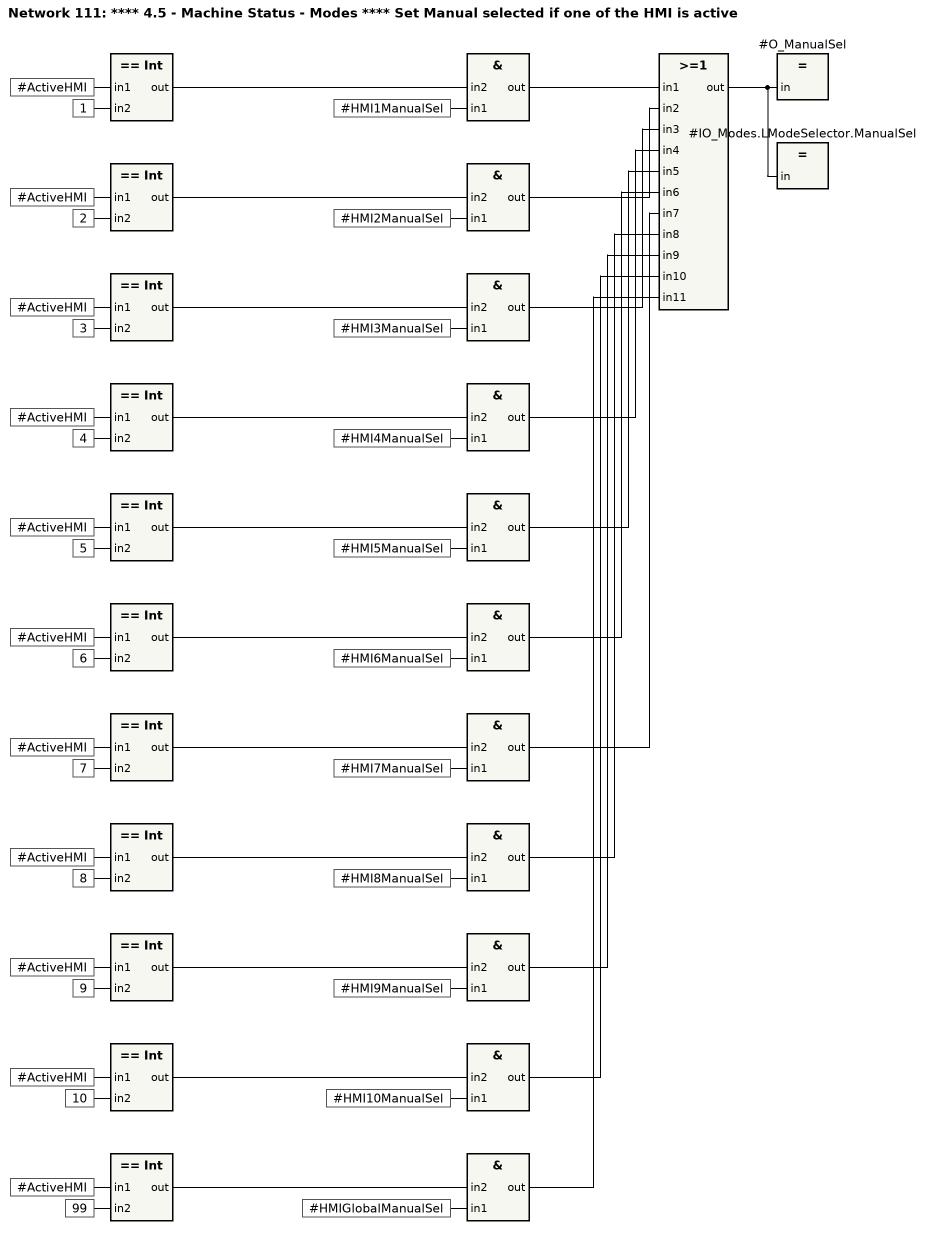
   #O_ManualSel := ((#ActiveHMI = 1) AND #HMI1ManualSel) OR ((#ActiveHMI = 2) AND #HMI2ManualSel) OR ((#ActiveHMI = 3) AND #HMI3ManualSel) OR ((#ActiveHMI = 4) AND #HMI4ManualSel) OR ((#ActiveHMI = 5) AND #HMI5ManualSel) OR ((#ActiveHMI = 6) AND #HMI6ManualSel) OR ((#ActiveHMI = 7) AND #HMI7ManualSel) OR ((#ActiveHMI = 8) AND #HMI8ManualSel) OR ((#ActiveHMI = 9) AND #HMI9ManualSel) OR ((#ActiveHMI = 10) AND #HMI10ManualSel) OR ((#ActiveHMI = 99) AND #HMIGlobalManualSel);
   #IO_Modes.LModeSelector.ManualSel := #O_ManualSel;
END_REGION

REGION Network 112: **** 4.6 - Machine Status - Indications **** Animation
   // Animation
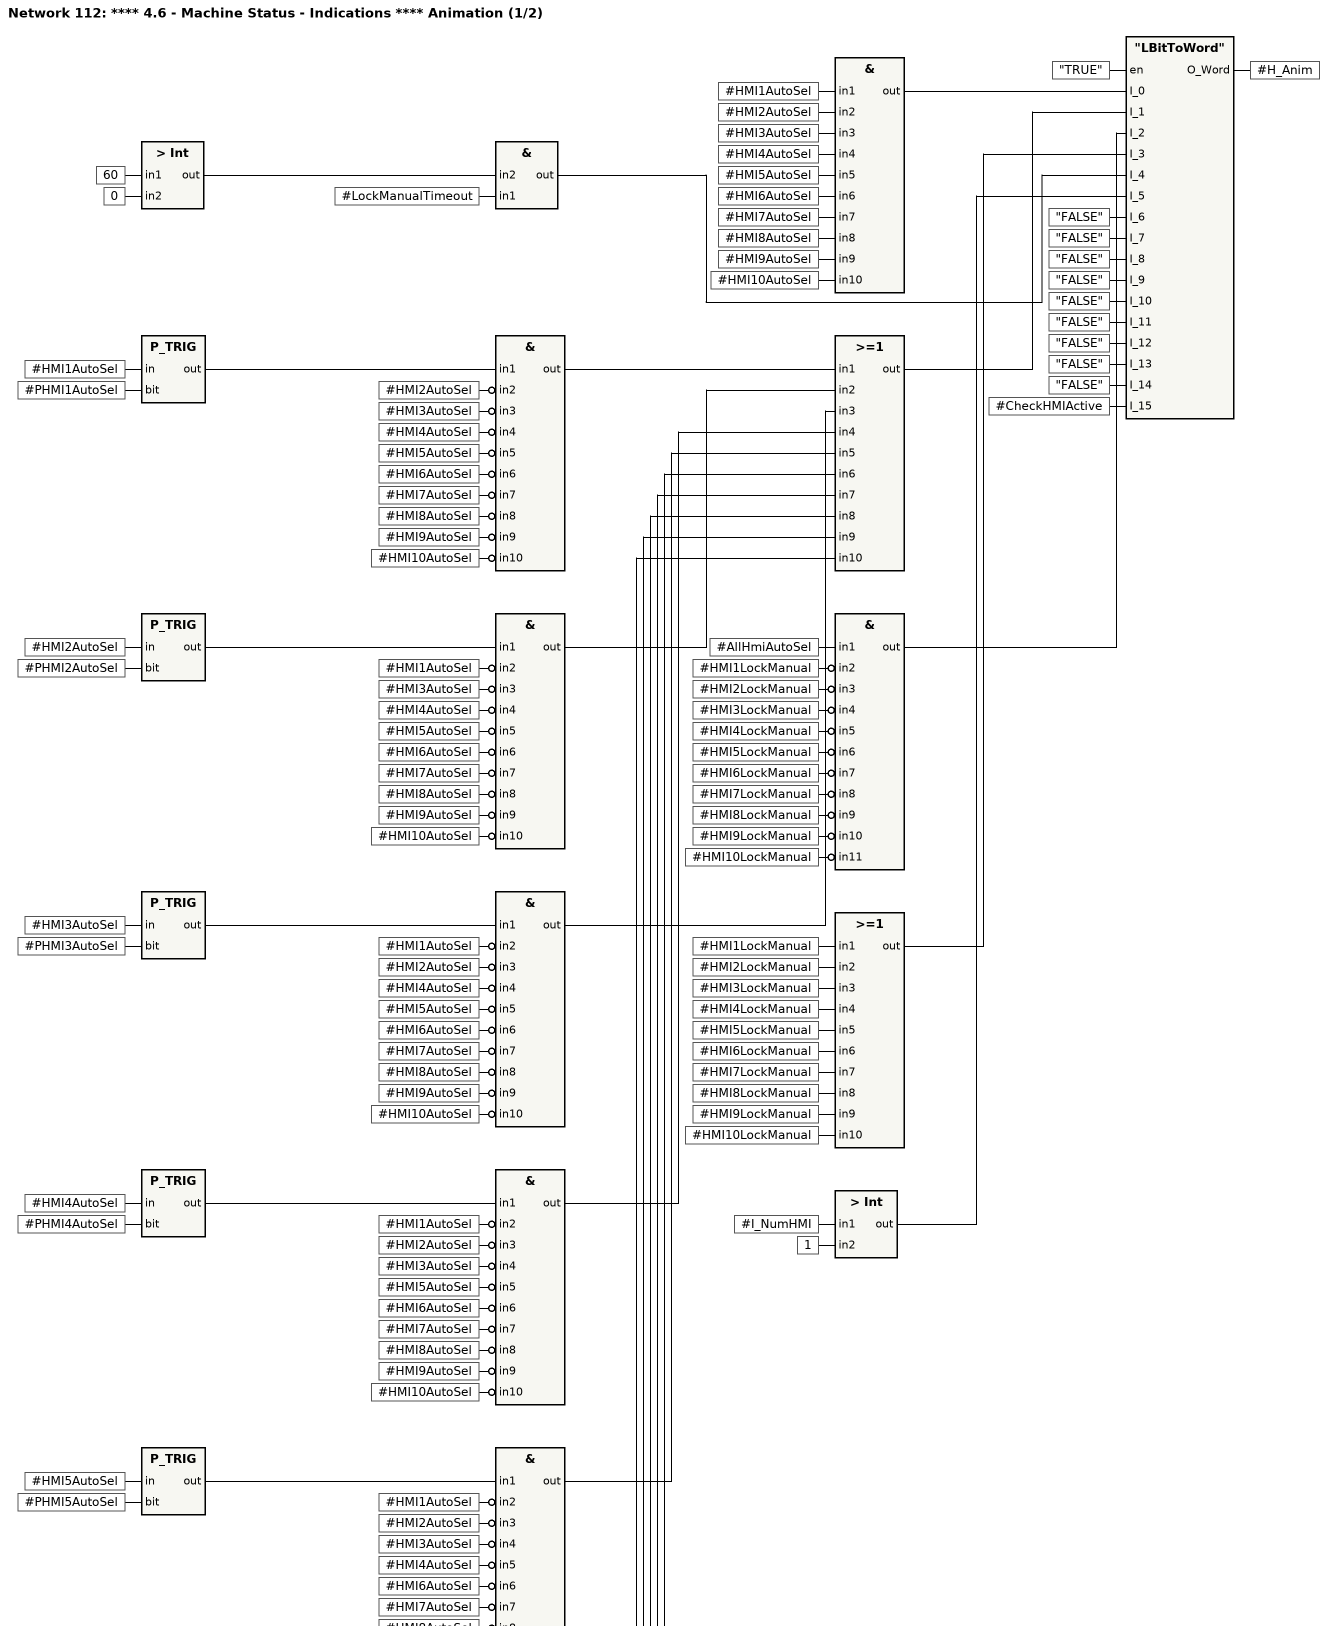
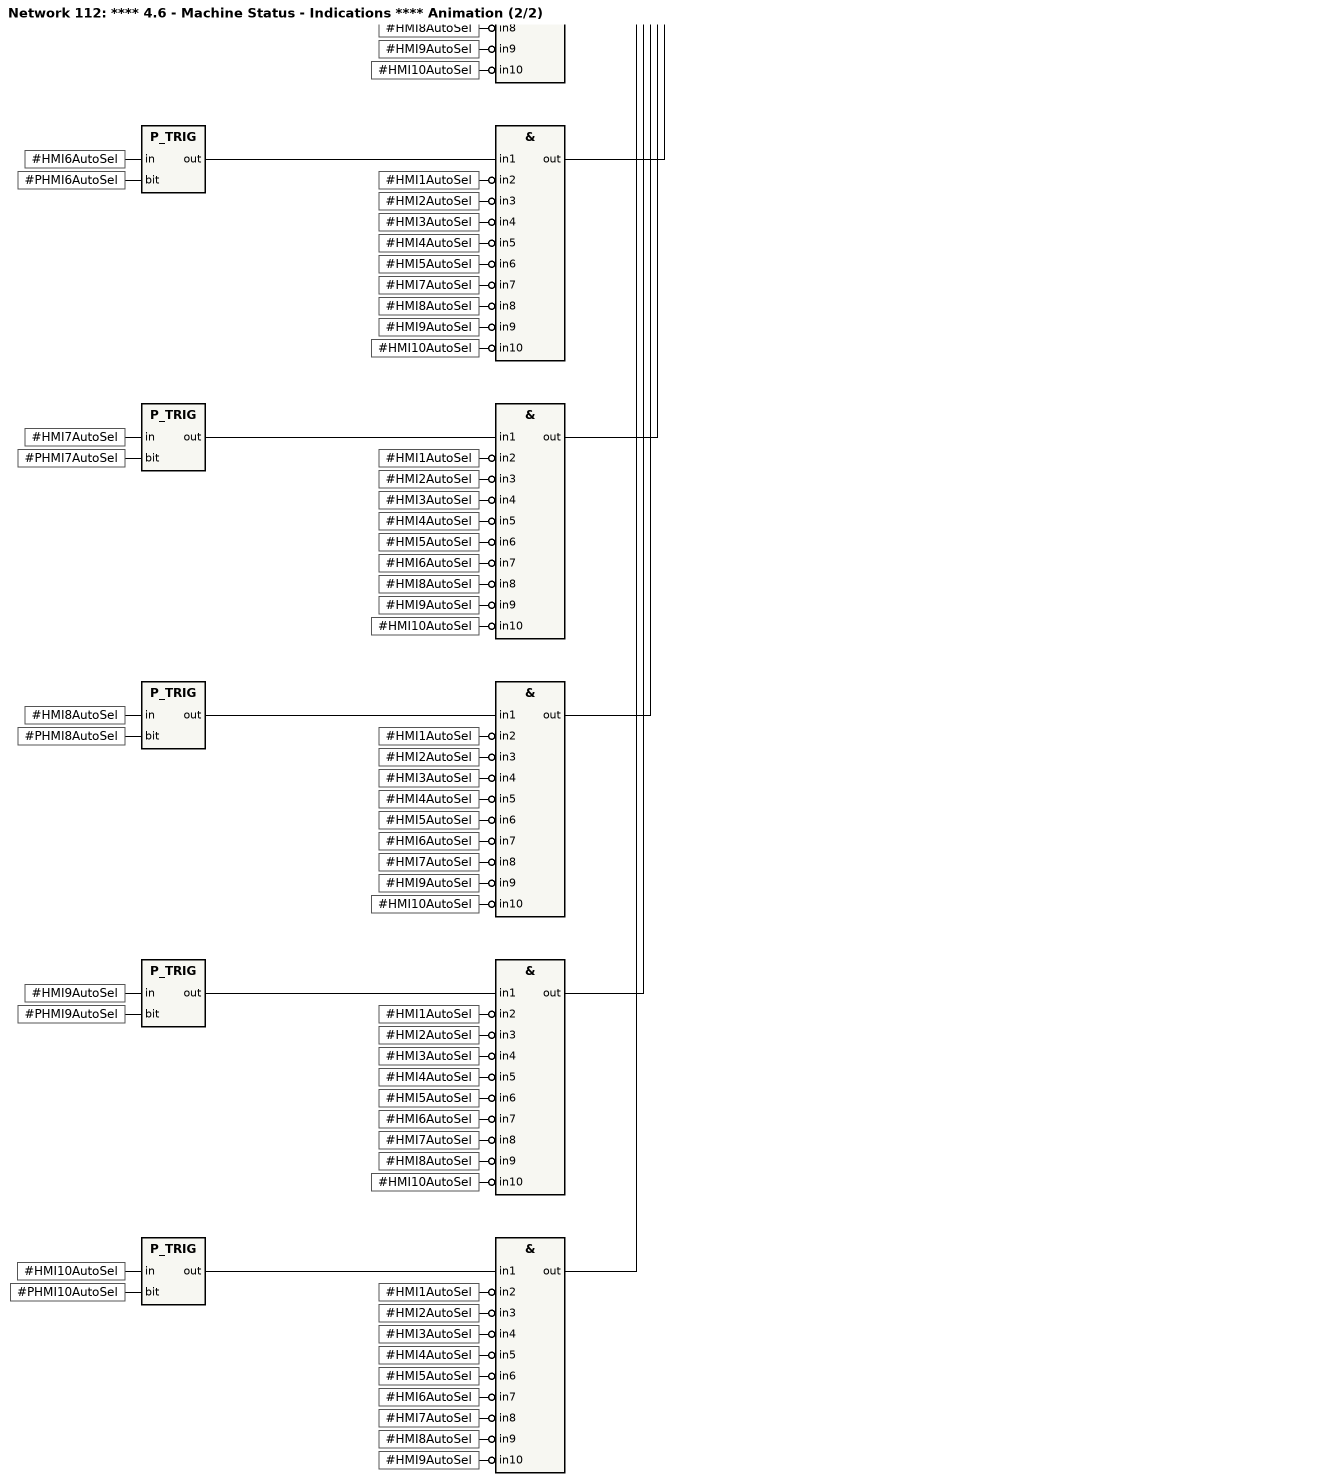
   #_w1 := #HMI1AutoSel AND NOT #PHMI1AutoSel;   // rising edge
   #PHMI1AutoSel := #HMI1AutoSel;
   #_w2 := #HMI2AutoSel AND NOT #PHMI2AutoSel;   // rising edge
   #PHMI2AutoSel := #HMI2AutoSel;
   #_w3 := #HMI3AutoSel AND NOT #PHMI3AutoSel;   // rising edge
   #PHMI3AutoSel := #HMI3AutoSel;
   #_w4 := #HMI4AutoSel AND NOT #PHMI4AutoSel;   // rising edge
   #PHMI4AutoSel := #HMI4AutoSel;
   #_w5 := #HMI5AutoSel AND NOT #PHMI5AutoSel;   // rising edge
   #PHMI5AutoSel := #HMI5AutoSel;
   #_w6 := #HMI6AutoSel AND NOT #PHMI6AutoSel;   // rising edge
   #PHMI6AutoSel := #HMI6AutoSel;
   #_w7 := #HMI7AutoSel AND NOT #PHMI7AutoSel;   // rising edge
   #PHMI7AutoSel := #HMI7AutoSel;
   #_w8 := #HMI8AutoSel AND NOT #PHMI8AutoSel;   // rising edge
   #PHMI8AutoSel := #HMI8AutoSel;
   #_w9 := #HMI9AutoSel AND NOT #PHMI9AutoSel;   // rising edge
   #PHMI9AutoSel := #HMI9AutoSel;
   #_w10 := #HMI10AutoSel AND NOT #PHMI10AutoSel;   // rising edge
   #PHMI10AutoSel := #HMI10AutoSel;
   IF "TRUE" THEN
       "LBitToWord"(I_0 := #HMI1AutoSel AND #HMI2AutoSel AND #HMI3AutoSel AND #HMI4AutoSel AND #HMI5AutoSel AND #HMI6AutoSel AND #HMI7AutoSel AND #HMI8AutoSel AND #HMI9AutoSel AND #HMI10AutoSel,
                    I_1 := (#_w1 AND NOT #HMI2AutoSel AND NOT #HMI3AutoSel AND NOT #HMI4AutoSel AND NOT #HMI5AutoSel AND NOT #HMI6AutoSel AND NOT #HMI7AutoSel AND NOT #HMI8AutoSel AND NOT #HMI9AutoSel AND NOT #HMI10AutoSel) OR (#_w2 AND NOT #HMI1AutoSel AND NOT #HMI3AutoSel AND NOT #HMI4AutoSel AND NOT #HMI5AutoSel AND NOT #HMI6AutoSel AND NOT #HMI7AutoSel AND NOT #HMI8AutoSel AND NOT #HMI9AutoSel AND NOT #HMI10AutoSel) OR (#_w3 AND NOT #HMI1AutoSel AND NOT #HMI2AutoSel AND NOT #HMI4AutoSel AND NOT #HMI5AutoSel AND NOT #HMI6AutoSel AND NOT #HMI7AutoSel AND NOT #HMI8AutoSel AND NOT #HMI9AutoSel AND NOT #HMI10AutoSel) OR (#_w4 AND NOT #HMI1AutoSel AND NOT #HMI2AutoSel AND NOT #HMI3AutoSel AND NOT #HMI5AutoSel AND NOT #HMI6AutoSel AND NOT #HMI7AutoSel AND NOT #HMI8AutoSel AND NOT #HMI9AutoSel AND NOT #HMI10AutoSel) OR (#_w5 AND NOT #HMI1AutoSel AND NOT #HMI2AutoSel AND NOT #HMI3AutoSel AND NOT #HMI4AutoSel AND NOT #HMI6AutoSel AND NOT #HMI7AutoSel AND NOT #HMI8AutoSel AND NOT #HMI9AutoSel AND NOT #HMI10AutoSel) OR (#_w6 AND NOT #HMI1AutoSel AND NOT #HMI2AutoSel AND NOT #HMI3AutoSel AND NOT #HMI4AutoSel AND NOT #HMI5AutoSel AND NOT #HMI7AutoSel AND NOT #HMI8AutoSel AND NOT #HMI9AutoSel AND NOT #HMI10AutoSel) OR (#_w7 AND NOT #HMI1AutoSel AND NOT #HMI2AutoSel AND NOT #HMI3AutoSel AND NOT #HMI4AutoSel AND NOT #HMI5AutoSel AND NOT #HMI6AutoSel AND NOT #HMI8AutoSel AND NOT #HMI9AutoSel AND NOT #HMI10AutoSel) OR (#_w8 AND NOT #HMI1AutoSel AND NOT #HMI2AutoSel AND NOT #HMI3AutoSel AND NOT #HMI4AutoSel AND NOT #HMI5AutoSel AND NOT #HMI6AutoSel AND NOT #HMI7AutoSel AND NOT #HMI9AutoSel AND NOT #HMI10AutoSel) OR (#_w9 AND NOT #HMI1AutoSel AND NOT #HMI2AutoSel AND NOT #HMI3AutoSel AND NOT #HMI4AutoSel AND NOT #HMI5AutoSel AND NOT #HMI6AutoSel AND NOT #HMI7AutoSel AND NOT #HMI8AutoSel AND NOT #HMI10AutoSel) OR (#_w10 AND NOT #HMI1AutoSel AND NOT #HMI2AutoSel AND NOT #HMI3AutoSel AND NOT #HMI4AutoSel AND NOT #HMI5AutoSel AND NOT #HMI6AutoSel AND NOT #HMI7AutoSel AND NOT #HMI8AutoSel AND NOT #HMI9AutoSel),
                    I_2 := #AllHmiAutoSel AND NOT #HMI1LockManual AND NOT #HMI2LockManual AND NOT #HMI3LockManual AND NOT #HMI4LockManual AND NOT #HMI5LockManual AND NOT #HMI6LockManual AND NOT #HMI7LockManual AND NOT #HMI8LockManual AND NOT #HMI9LockManual AND NOT #HMI10LockManual,
                    I_3 := #HMI1LockManual OR #HMI2LockManual OR #HMI3LockManual OR #HMI4LockManual OR #HMI5LockManual OR #HMI6LockManual OR #HMI7LockManual OR #HMI8LockManual OR #HMI9LockManual OR #HMI10LockManual,
                    I_4 := (60 > 0) AND #LockManualTimeout,
                    I_5 := #I_NumHMI > 1,
                    I_6 := "FALSE",
                    I_7 := "FALSE",
                    I_8 := "FALSE",
                    I_9 := "FALSE",
                    I_10 := "FALSE",
                    I_11 := "FALSE",
                    I_12 := "FALSE",
                    I_13 := "FALSE",
                    I_14 := "FALSE",
                    I_15 := #CheckHMIActive,
                    O_Word => #H_Anim);
   END_IF;
END_REGION

REGION Network 113: **** 5.2 - Equations - Flow **** Reset transport memory on active HMI
   // Reset transport memory on active HMI
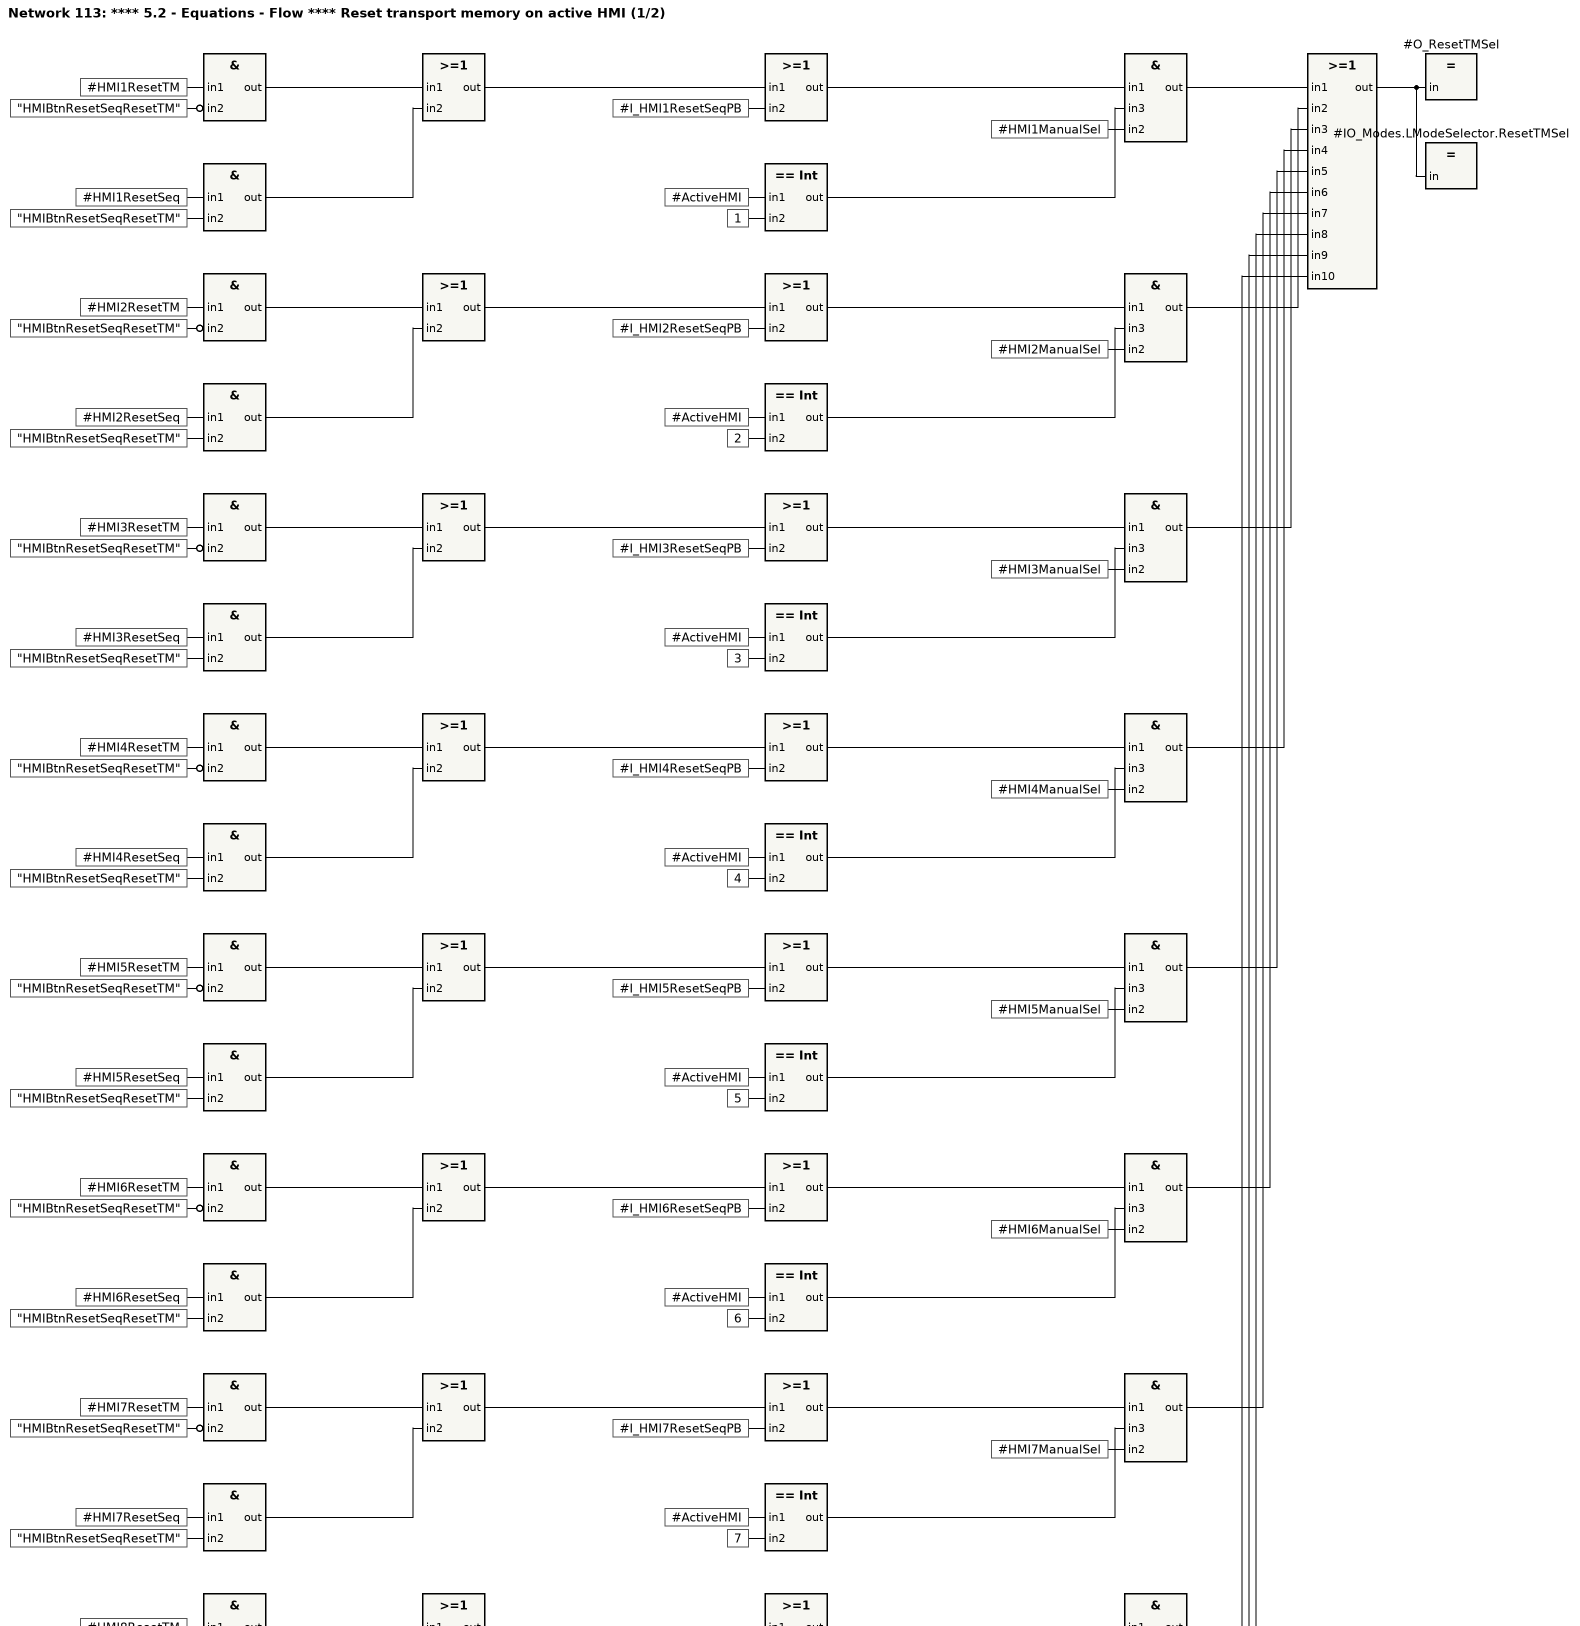
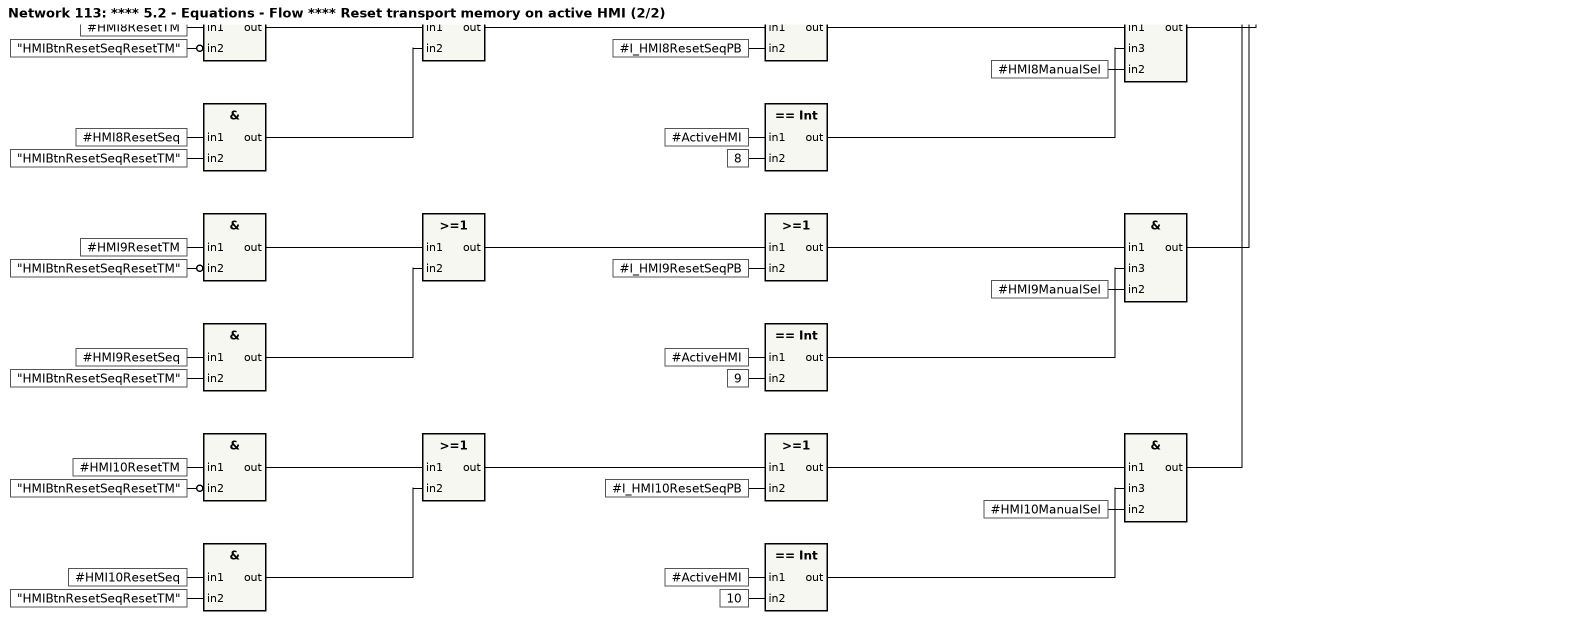
   #O_ResetTMSel := (((#HMI1ResetTM AND NOT "HMIBtnResetSeqResetTM") OR (#HMI1ResetSeq AND "HMIBtnResetSeqResetTM") OR #I_HMI1ResetSeqPB) AND (#ActiveHMI = 1) AND #HMI1ManualSel) OR (((#HMI2ResetTM AND NOT "HMIBtnResetSeqResetTM") OR (#HMI2ResetSeq AND "HMIBtnResetSeqResetTM") OR #I_HMI2ResetSeqPB) AND (#ActiveHMI = 2) AND #HMI2ManualSel) OR (((#HMI3ResetTM AND NOT "HMIBtnResetSeqResetTM") OR (#HMI3ResetSeq AND "HMIBtnResetSeqResetTM") OR #I_HMI3ResetSeqPB) AND (#ActiveHMI = 3) AND #HMI3ManualSel) OR (((#HMI4ResetTM AND NOT "HMIBtnResetSeqResetTM") OR (#HMI4ResetSeq AND "HMIBtnResetSeqResetTM") OR #I_HMI4ResetSeqPB) AND (#ActiveHMI = 4) AND #HMI4ManualSel) OR (((#HMI5ResetTM AND NOT "HMIBtnResetSeqResetTM") OR (#HMI5ResetSeq AND "HMIBtnResetSeqResetTM") OR #I_HMI5ResetSeqPB) AND (#ActiveHMI = 5) AND #HMI5ManualSel) OR (((#HMI6ResetTM AND NOT "HMIBtnResetSeqResetTM") OR (#HMI6ResetSeq AND "HMIBtnResetSeqResetTM") OR #I_HMI6ResetSeqPB) AND (#ActiveHMI = 6) AND #HMI6ManualSel) OR (((#HMI7ResetTM AND NOT "HMIBtnResetSeqResetTM") OR (#HMI7ResetSeq AND "HMIBtnResetSeqResetTM") OR #I_HMI7ResetSeqPB) AND (#ActiveHMI = 7) AND #HMI7ManualSel) OR (((#HMI8ResetTM AND NOT "HMIBtnResetSeqResetTM") OR (#HMI8ResetSeq AND "HMIBtnResetSeqResetTM") OR #I_HMI8ResetSeqPB) AND (#ActiveHMI = 8) AND #HMI8ManualSel) OR (((#HMI9ResetTM AND NOT "HMIBtnResetSeqResetTM") OR (#HMI9ResetSeq AND "HMIBtnResetSeqResetTM") OR #I_HMI9ResetSeqPB) AND (#ActiveHMI = 9) AND #HMI9ManualSel) OR (((#HMI10ResetTM AND NOT "HMIBtnResetSeqResetTM") OR (#HMI10ResetSeq AND "HMIBtnResetSeqResetTM") OR #I_HMI10ResetSeqPB) AND (#ActiveHMI = 10) AND #HMI10ManualSel);
   #IO_Modes.LModeSelector.ResetTMSel := #O_ResetTMSel;
END_REGION

REGION Network 114: **** 5.2 - Equations - Flow **** Reset sequence on active HMI
   // Reset sequence on active HMI
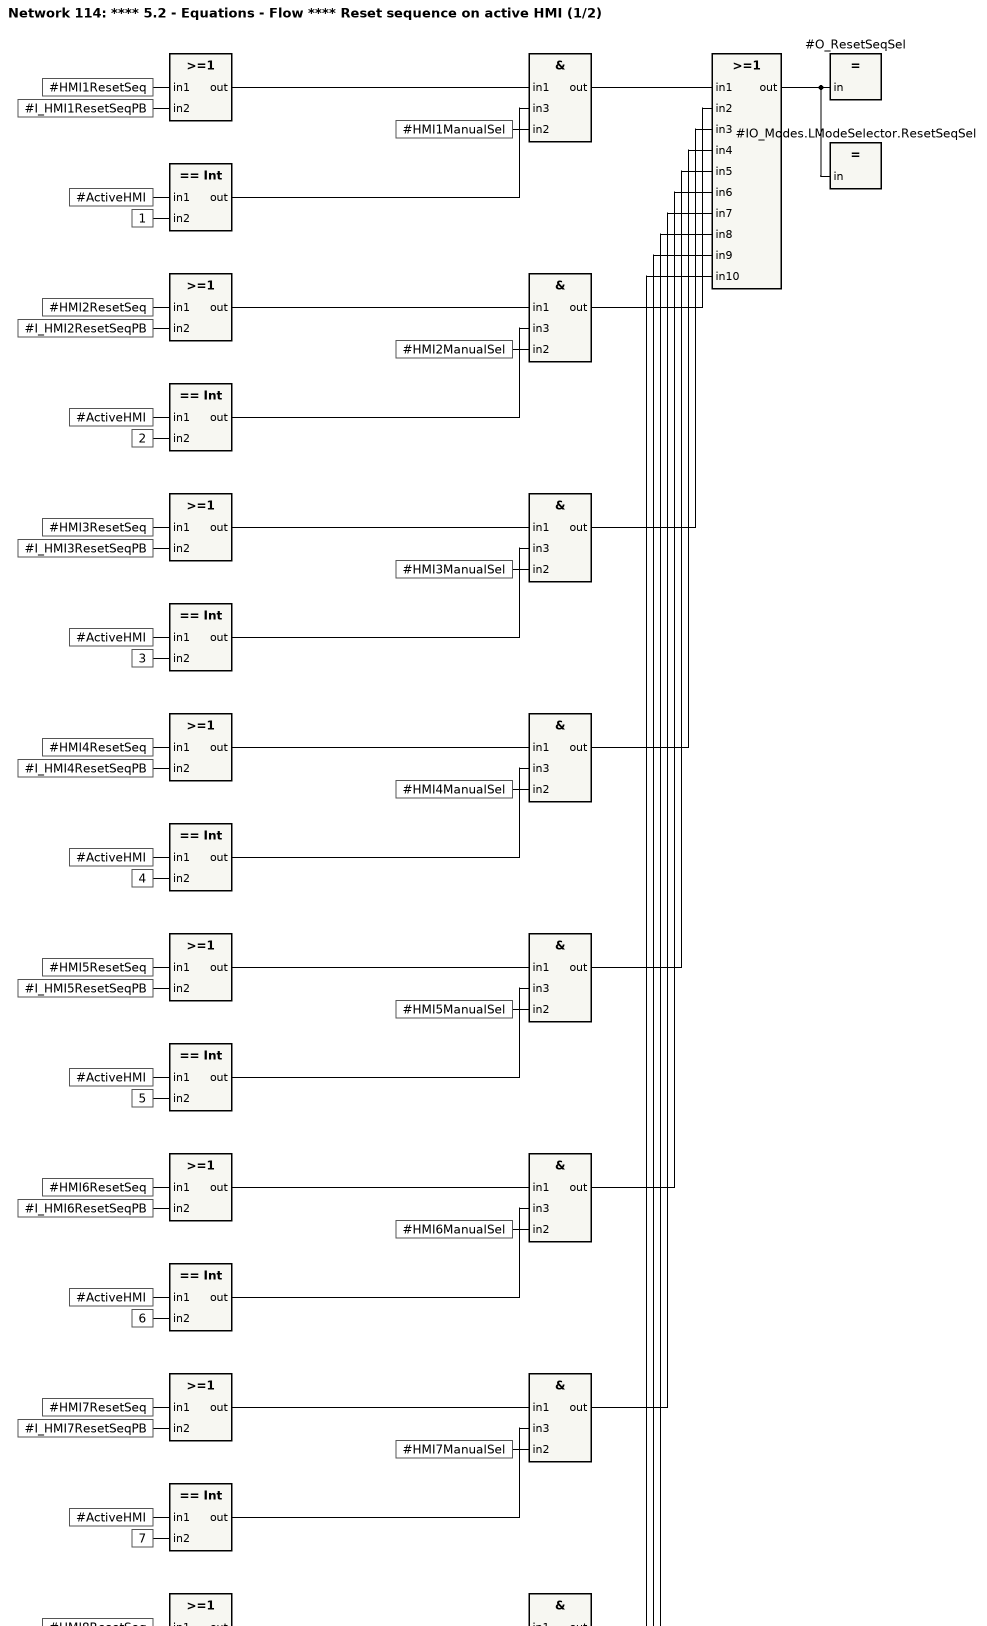
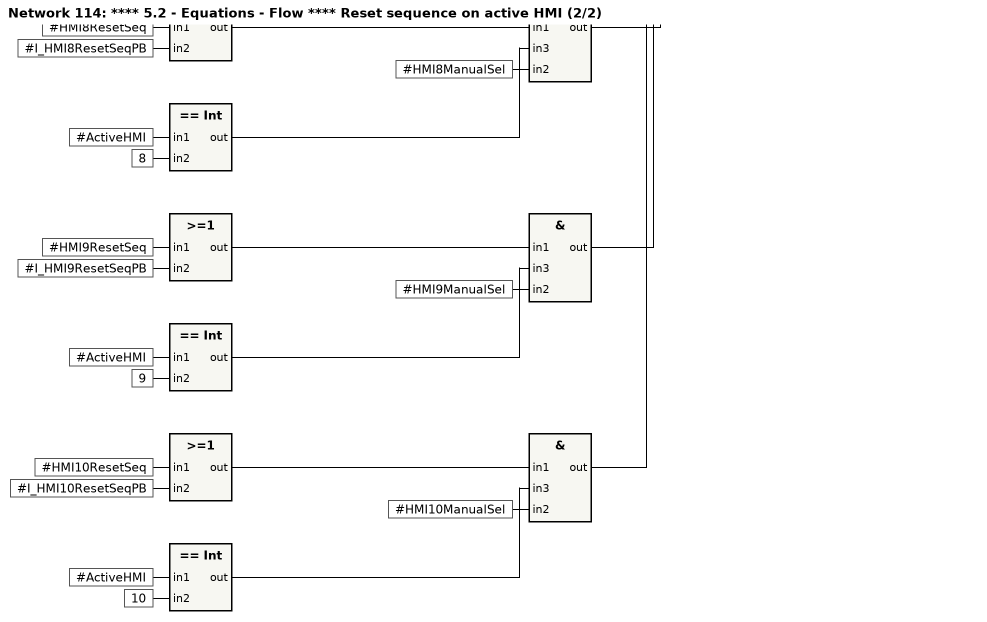
   #O_ResetSeqSel := ((#HMI1ResetSeq OR #I_HMI1ResetSeqPB) AND (#ActiveHMI = 1) AND #HMI1ManualSel) OR ((#HMI2ResetSeq OR #I_HMI2ResetSeqPB) AND (#ActiveHMI = 2) AND #HMI2ManualSel) OR ((#HMI3ResetSeq OR #I_HMI3ResetSeqPB) AND (#ActiveHMI = 3) AND #HMI3ManualSel) OR ((#HMI4ResetSeq OR #I_HMI4ResetSeqPB) AND (#ActiveHMI = 4) AND #HMI4ManualSel) OR ((#HMI5ResetSeq OR #I_HMI5ResetSeqPB) AND (#ActiveHMI = 5) AND #HMI5ManualSel) OR ((#HMI6ResetSeq OR #I_HMI6ResetSeqPB) AND (#ActiveHMI = 6) AND #HMI6ManualSel) OR ((#HMI7ResetSeq OR #I_HMI7ResetSeqPB) AND (#ActiveHMI = 7) AND #HMI7ManualSel) OR ((#HMI8ResetSeq OR #I_HMI8ResetSeqPB) AND (#ActiveHMI = 8) AND #HMI8ManualSel) OR ((#HMI9ResetSeq OR #I_HMI9ResetSeqPB) AND (#ActiveHMI = 9) AND #HMI9ManualSel) OR ((#HMI10ResetSeq OR #I_HMI10ResetSeqPB) AND (#ActiveHMI = 10) AND #HMI10ManualSel);
   #IO_Modes.LModeSelector.ResetSeqSel := #O_ResetSeqSel;
END_REGION

REGION Network 115: **** 5.2 - Equations - Flow **** Check Active HMI again - HMI <> 0
   // Check Active HMI again
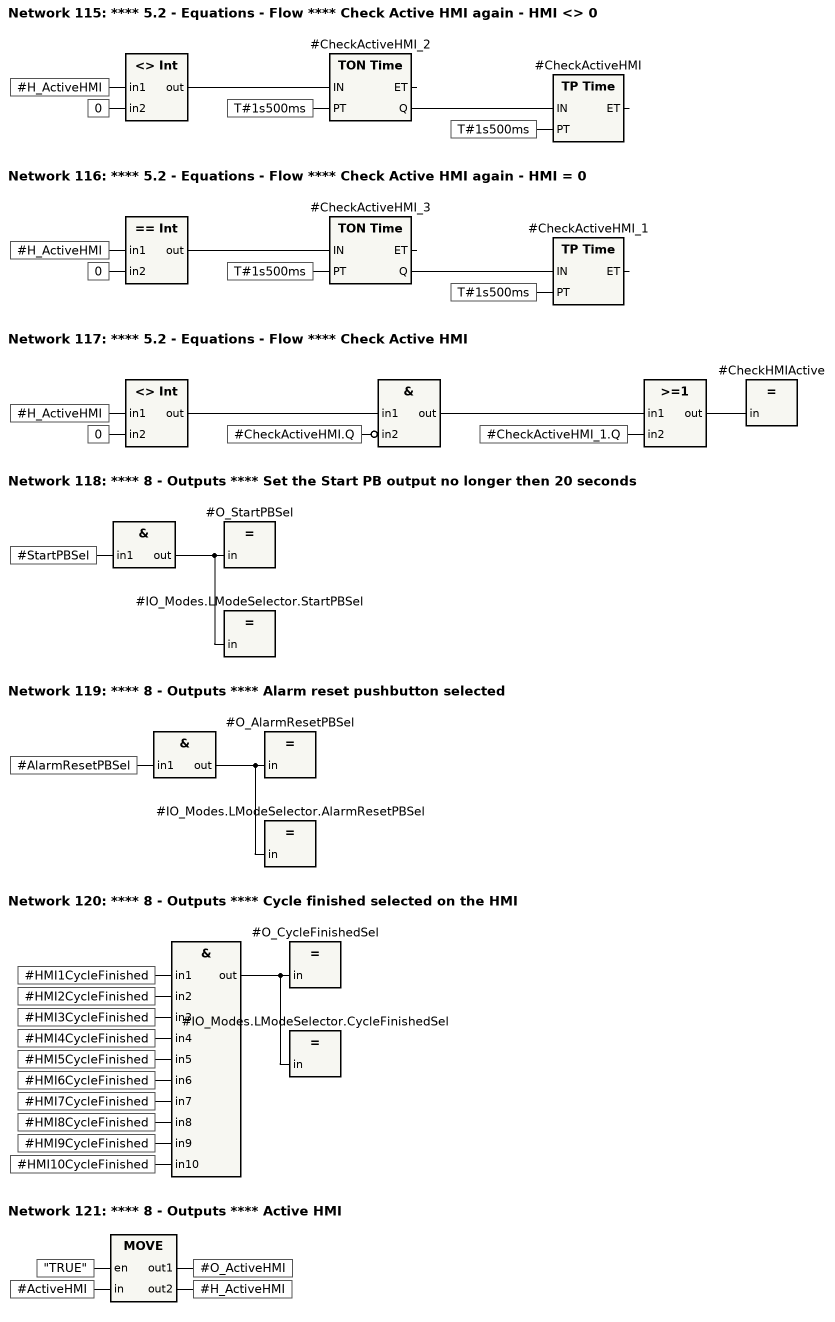
   #CheckActiveHMI_2(IN := #H_ActiveHMI <> 0, PT := T#1s500ms);   // TON
   #CheckActiveHMI(IN := #CheckActiveHMI_2.Q, PT := T#1s500ms);   // TP
END_REGION

REGION Network 116: **** 5.2 - Equations - Flow **** Check Active HMI again - HMI = 0
   // Check Active HMI again
   #CheckActiveHMI_3(IN := #H_ActiveHMI = 0, PT := T#1s500ms);   // TON
   #CheckActiveHMI_1(IN := #CheckActiveHMI_3.Q, PT := T#1s500ms);   // TP
END_REGION

REGION Network 117: **** 5.2 - Equations - Flow **** Check Active HMI
   // Check Active HMI
   #CheckHMIActive := ((#H_ActiveHMI <> 0) AND NOT #CheckActiveHMI.Q) OR #CheckActiveHMI_1.Q;
END_REGION

REGION Network 118: **** 8 - Outputs **** Set the Start PB output no longer then 20 seconds
   // Set the Start PB output no longer then 20 seconds
   #O_StartPBSel := #StartPBSel;
   #IO_Modes.LModeSelector.StartPBSel := #StartPBSel;
END_REGION

REGION Network 119: **** 8 - Outputs **** Alarm reset pushbutton selected
   // Alarm reset pushbutton selected
   #O_AlarmResetPBSel := #AlarmResetPBSel;
   #IO_Modes.LModeSelector.AlarmResetPBSel := #AlarmResetPBSel;
END_REGION

REGION Network 120: **** 8 - Outputs **** Cycle finished selected on the HMI
   // Cycle finished selected on the HMI
   #O_CycleFinishedSel := #HMI1CycleFinished AND #HMI2CycleFinished AND #HMI3CycleFinished AND #HMI4CycleFinished AND #HMI5CycleFinished AND #HMI6CycleFinished AND #HMI7CycleFinished AND #HMI8CycleFinished AND #HMI9CycleFinished AND #HMI10CycleFinished;
   #IO_Modes.LModeSelector.CycleFinishedSel := #O_CycleFinishedSel;
END_REGION

REGION Network 121: **** 8 - Outputs **** Active HMI
   // Active HMI
   IF "TRUE" THEN
       #O_ActiveHMI := #ActiveHMI;
       #H_ActiveHMI := #ActiveHMI;
   END_IF;
END_REGION

REGION Network 122: **** 8 - Outputs **** Lock Manual Time
   // Lock Manual Time
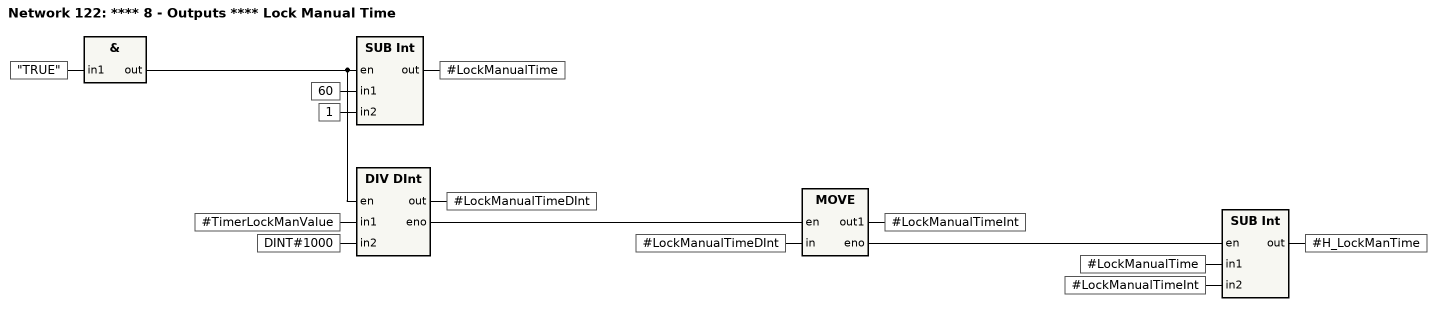
   // ENO of a box is taken as its EN; it also drops when the box reports an error
   IF "TRUE" THEN
       #LockManualTime := 60 - 1;
       #LockManualTimeDInt := #TimerLockManValue / DINT#1000;
       #LockManualTimeInt := #LockManualTimeDInt;
       #H_LockManTime := #LockManualTime - #LockManualTimeInt;
   END_IF;
END_REGION
END_FUNCTION_BLOCK

FUNCTION_BLOCK "LHMIResetStart"   // FB1006, FBD
TITLE = LHMIResetStart
{ S7_Optimized_Access := 'FALSE' }
AUTHOR : VCC
FAMILY : Control
NAME : ModeSel
VERSION : 1.0
// ================================================================================
// This module is creating the needed integers for the F_ACK_OP module from reset 
// and start selections made on the HMI.  It also foresees the outputs for reset 
// and start to be connected to the modeselector.
// ================================================================================
// stored: AutoNumber false, IsIECCheckEnabled false, SetENOAutomatically False, UDAEnableTagReadback false
   VAR_INPUT
      I_SafetyNotOk { ExternalAccessible := 'False'; ExternalVisible := 'False'; ExternalWritable := 'False'} : Bool;   // Safety is not ok
      I_FailSafeResetAck { ExternalAccessible := 'False'; ExternalVisible := 'False'; ExternalWritable := 'False'} : Bool;   // F_Ack_Op FB in safety program is requesting value 9 on FailSafeReset output
      I_FailSafeAckID { ExternalAccessible := 'False'; ExternalVisible := 'False'; ExternalWritable := 'False'} : Int;   // F_Ack ID
   END_VAR
   VAR_OUTPUT
      O_HMIAlarmResetPBSel { ExternalAccessible := 'False'; ExternalVisible := 'False'; ExternalWritable := 'False'} : Bool;   // Alarm reset is activated
      O_HMIStartPBSel { ExternalAccessible := 'False'; ExternalVisible := 'False'; ExternalWritable := 'False'} : Bool;   // Start is activated
   END_VAR
   VAR_IN_OUT
      H_HMI1ModeCmd { ExternalAccessible := 'False'; ExternalVisible := 'False'; ExternalWritable := 'False'} : Word;   // Mode commands from HMI1
      IO_FailsafeReset { ExternalAccessible := 'False'; ExternalVisible := 'False'; ExternalWritable := 'False'} : Int;   // Number to Failsafe to reset safety
   END_VAR
   VAR DB_SPECIFIC
      HMI1Start { ExternalAccessible := 'False'; ExternalVisible := 'False'; ExternalWritable := 'False'} : Bool;   // Start on HMI1
      HMI1AlarmReset { ExternalAccessible := 'False'; ExternalVisible := 'False'; ExternalWritable := 'False'} : Bool;   // AlarmReset on HMI1
      HMI1AlarmResetAck { ExternalAccessible := 'False'; ExternalVisible := 'False'; ExternalWritable := 'False'} : Bool;   // Alarm Reset acknowledge from HMI1
      HMIAlarmResetPBSel { ExternalAccessible := 'False'; ExternalVisible := 'False'; ExternalWritable := 'False'} : Bool;   // Alarm reset is activated
      HMIStartPE { ExternalAccessible := 'False'; ExternalVisible := 'False'; ExternalWritable := 'False'} : Bool;   // Positive edge on start button from HMI
      HMIAlarmResetAckPE { ExternalAccessible := 'False'; ExternalVisible := 'False'; ExternalWritable := 'False'} : Bool;   // Positive edge on AlarmResetAck button from HMI
      AlarmResetPBSelReset { ExternalAccessible := 'False'; ExternalVisible := 'False'; ExternalWritable := 'False'} : Bool;   // Reset AlarmResetPBSel after predefined time
      AlarmResetPBSelResetPE { ExternalAccessible := 'False'; ExternalVisible := 'False'; ExternalWritable := 'False'} : Bool;   // Positive edge of AlarmResetPbSelReset
      FailSafeReset6Pulse { ExternalAccessible := 'False'; ExternalVisible := 'False'; ExternalWritable := 'False'} : Bool;   // Pulse to set value 6 on FailSafeReset Output
      FailSafeReset9Pulse { ExternalAccessible := 'False'; ExternalVisible := 'False'; ExternalWritable := 'False'} : Bool;   // Pulse to set value 9 on FailSafeReset Output
      ResetAlarmAckMemPulse { ExternalAccessible := 'False'; ExternalVisible := 'False'; ExternalWritable := 'False'} : Bool;   // Pulse to reset AlarmResetAckMem on negative edge of I_FailSafeResetAck
      AlarmResetAckMem { ExternalAccessible := 'False'; ExternalVisible := 'False'; ExternalWritable := 'False'} : Bool;   // memory : Pushbutton AlarmResetAck has been pushed on HMI
      FailsafeReset { ExternalAccessible := 'False'; ExternalVisible := 'False'; ExternalWritable := 'False'} : Int;   // Number to Failsafe to reset safety
   END_VAR
   VAR
      TimerAlarmResetPB { ExternalAccessible := 'False'; ExternalVisible := 'False'; ExternalWritable := 'False'} : "LTimer";
   END_VAR
   VAR_TEMP   // added for the SCL form of the ladder/FBD networks
      _w1 : Bool;
      _w2 : Bool;
   END_VAR
BEGIN

REGION Network 1: **** 1 - Inputs **** Extract the modeselection from HMI 1
   // Extract the modeselection from HMI 1
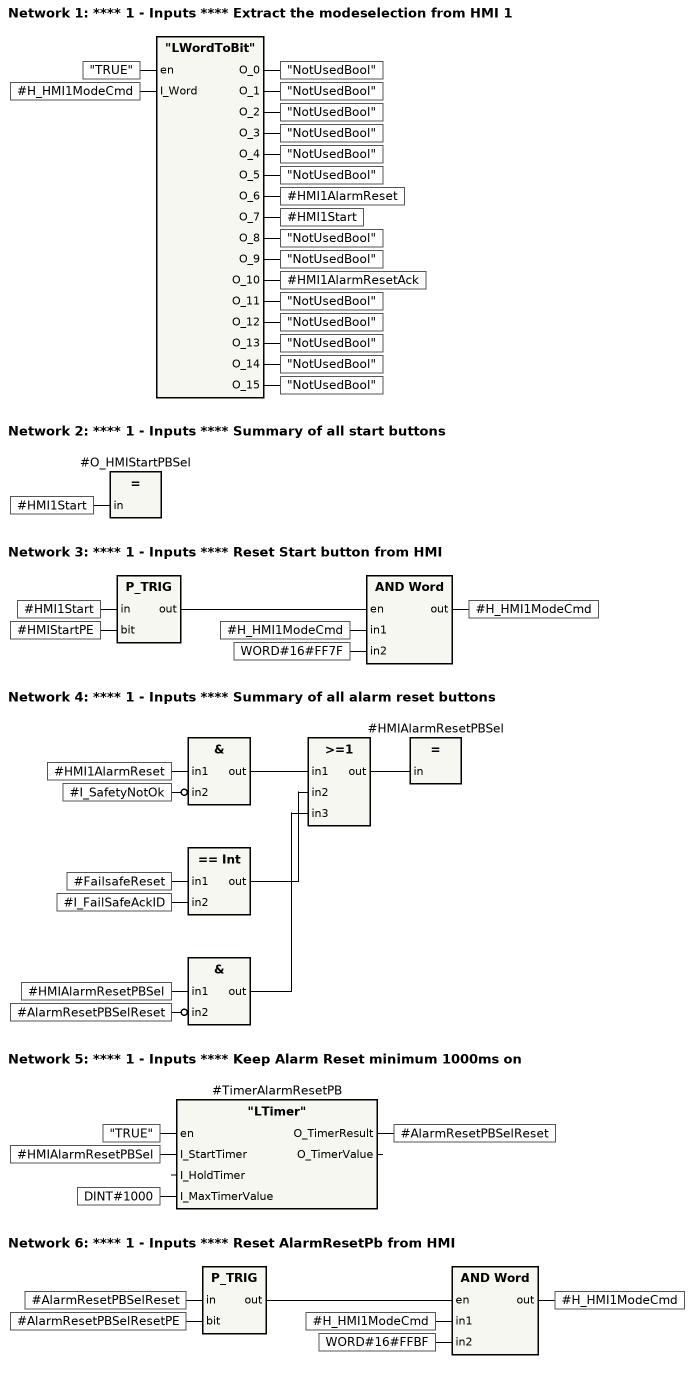
   IF "TRUE" THEN
       "LWordToBit"(I_Word := #H_HMI1ModeCmd,
                    O_0 => "NotUsedBool",
                    O_1 => "NotUsedBool",
                    O_2 => "NotUsedBool",
                    O_3 => "NotUsedBool",
                    O_4 => "NotUsedBool",
                    O_5 => "NotUsedBool",
                    O_6 => #HMI1AlarmReset,
                    O_7 => #HMI1Start,
                    O_8 => "NotUsedBool",
                    O_9 => "NotUsedBool",
                    O_10 => #HMI1AlarmResetAck,
                    O_11 => "NotUsedBool",
                    O_12 => "NotUsedBool",
                    O_13 => "NotUsedBool",
                    O_14 => "NotUsedBool",
                    O_15 => "NotUsedBool");
   END_IF;
END_REGION

REGION Network 2: **** 1 - Inputs **** Summary of all start buttons
   // Summary of all start buttons
   #O_HMIStartPBSel := #HMI1Start;
END_REGION

REGION Network 3: **** 1 - Inputs **** Reset Start button from HMI
   // Reset Start button from HMI
   #_w1 := #HMI1Start AND NOT #HMIStartPE;   // rising edge
   #HMIStartPE := #HMI1Start;
   IF #_w1 THEN #H_HMI1ModeCmd := #H_HMI1ModeCmd AND WORD#16#FF7F; END_IF;
END_REGION

REGION Network 4: **** 1 - Inputs **** Summary of all alarm reset buttons
   // Summary of all alarm reset buttons
   #HMIAlarmResetPBSel := (#HMI1AlarmReset AND NOT #I_SafetyNotOk) OR (#FailsafeReset = #I_FailSafeAckID) OR (#HMIAlarmResetPBSel AND NOT #AlarmResetPBSelReset);
END_REGION

REGION Network 5: **** 1 - Inputs **** Keep Alarm Reset minimum 1000ms on
   // Keep Alarm Reset minimum 1000ms on
   IF "TRUE" THEN
       #TimerAlarmResetPB(I_StartTimer := #HMIAlarmResetPBSel,   // "LTimer"
                          I_MaxTimerValue := DINT#1000,
                          O_TimerResult => #AlarmResetPBSelReset);
   END_IF;
END_REGION

REGION Network 6: **** 1 - Inputs **** Reset AlarmResetPb from HMI
   // Reset AlarmResetPb from HMI
   #_w1 := #AlarmResetPBSelReset AND NOT #AlarmResetPBSelResetPE;   // rising edge
   #AlarmResetPBSelResetPE := #AlarmResetPBSelReset;
   IF #_w1 THEN #H_HMI1ModeCmd := #H_HMI1ModeCmd AND WORD#16#FFBF; END_IF;
END_REGION

REGION Network 7: **** 1 - Inputs **** Reset AlarmResetAckPb from HMI
   // Reset AlarmResetAckPb from HMI
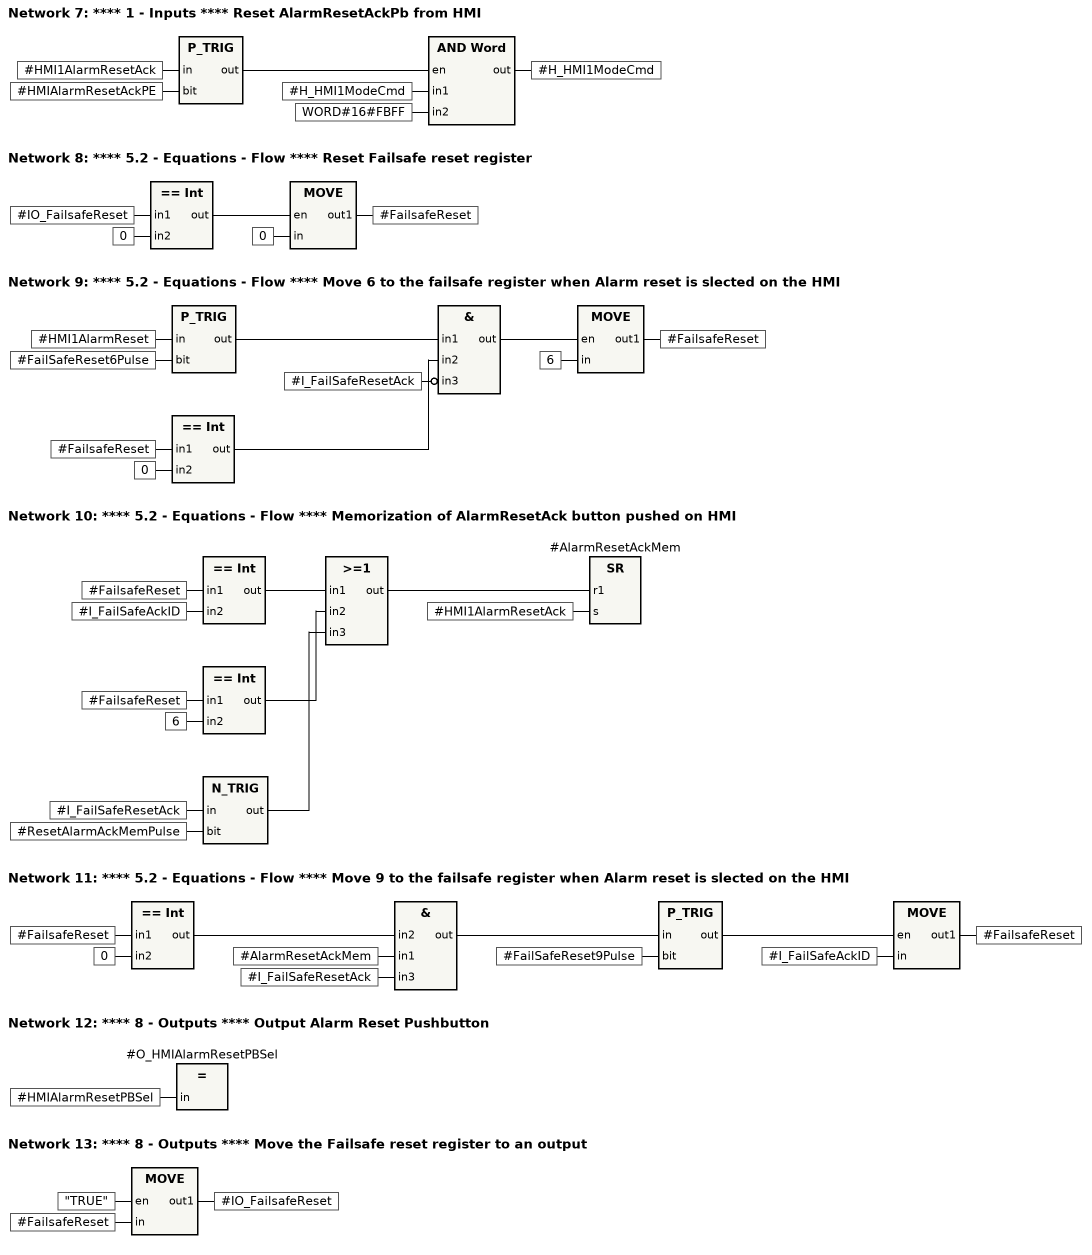
   #_w1 := #HMI1AlarmResetAck AND NOT #HMIAlarmResetAckPE;   // rising edge
   #HMIAlarmResetAckPE := #HMI1AlarmResetAck;
   IF #_w1 THEN #H_HMI1ModeCmd := #H_HMI1ModeCmd AND WORD#16#FBFF; END_IF;
END_REGION

REGION Network 8: **** 5.2 - Equations - Flow **** Reset Failsafe reset register
   // Reset Failsafe reset register
   IF #IO_FailsafeReset = 0 THEN #FailsafeReset := 0; END_IF;
END_REGION

REGION Network 9: **** 5.2 - Equations - Flow **** Move 6 to the failsafe register when Alarm reset is slected on the HMI
   // Move 6 to the failsafe register when Alarm reset is slected on the HMI
   #_w1 := #HMI1AlarmReset AND NOT #FailSafeReset6Pulse;   // rising edge
   #FailSafeReset6Pulse := #HMI1AlarmReset;
   IF #_w1 AND (#FailsafeReset = 0) AND NOT #I_FailSafeResetAck THEN #FailsafeReset := 6; END_IF;
END_REGION

REGION Network 10: **** 5.2 - Equations - Flow **** Memorization of AlarmResetAck button pushed on HMI
   // Memorization of AlarmResetAck button pushed on HMI
   #_w1 := NOT #I_FailSafeResetAck AND #ResetAlarmAckMemPulse;   // falling edge
   #ResetAlarmAckMemPulse := #I_FailSafeResetAck;
   IF #HMI1AlarmResetAck THEN
       #AlarmResetAckMem := TRUE;   // SR flip-flop
   END_IF;
   IF (#FailsafeReset = #I_FailSafeAckID) OR (#FailsafeReset = 6) OR #_w1 THEN
       #AlarmResetAckMem := FALSE;
   END_IF;
END_REGION

REGION Network 11: **** 5.2 - Equations - Flow **** Move 9 to the failsafe register when Alarm reset is slected on the HMI
   // Move 9 to the failsafe register when Alarm reset is slected on the HMI
   #_w1 := (#FailsafeReset = 0) AND #AlarmResetAckMem AND #I_FailSafeResetAck;
   #_w2 := #_w1 AND NOT #FailSafeReset9Pulse;   // rising edge
   #FailSafeReset9Pulse := #_w1;
   IF #_w2 THEN #FailsafeReset := #I_FailSafeAckID; END_IF;
END_REGION

REGION Network 12: **** 8 - Outputs **** Output Alarm Reset Pushbutton
   // Output Alarm Reset Pushbutton
   #O_HMIAlarmResetPBSel := #HMIAlarmResetPBSel;
END_REGION

REGION Network 13: **** 8 - Outputs **** Move the Failsafe reset register to an output
   // Move the Failsafe reset register to an output
   IF "TRUE" THEN #IO_FailsafeReset := #FailsafeReset; END_IF;
END_REGION
END_FUNCTION_BLOCK

FUNCTION_BLOCK "LGenHooterFlash"   // FB1007, FBD
TITLE = LGenHootFlash
{ S7_Optimized_Access := 'FALSE' }
AUTHOR : VCG
FAMILY : VCGGen
VERSION : 1.0
// ==============================================================================
// FB 
// ==============================================================================
// stored: AutoNumber false, IsIECCheckEnabled false, SetENOAutomatically False, UDAEnableTagReadback false
   VAR_INPUT
      I_Lamptest { ExternalAccessible := 'False'; ExternalVisible := 'False'; ExternalWritable := 'False'} : Bool;   // Summation of lamptest buttons
      I_GenResetAlarm { ExternalAccessible := 'False'; ExternalVisible := 'False'; ExternalWritable := 'False'} : Bool;   // General reset alarm
      I_GenAlarmA { ExternalAccessible := 'False'; ExternalVisible := 'False'; ExternalWritable := 'False'} : Bool;   // General Alarm A active
      I_GenAlarmB { ExternalAccessible := 'False'; ExternalVisible := 'False'; ExternalWritable := 'False'} : Bool;   // General Alarm B active
      I_GenAlarmC { ExternalAccessible := 'False'; ExternalVisible := 'False'; ExternalWritable := 'False'} : Bool;   // General Alarm C active
      I_HardwareAlarm { ExternalAccessible := 'False'; ExternalVisible := 'False'; ExternalWritable := 'False'} : Bool;   // Safety circuit hardware Alarm active
      I_GenWarningStart { ExternalAccessible := 'False'; ExternalVisible := 'False'; ExternalWritable := 'False'} : Bool;   // Warning start from station
   END_VAR
   VAR_OUTPUT
      O_HooterAK { ExternalAccessible := 'False'; ExternalVisible := 'False'; ExternalWritable := 'False'} : Bool;   // Steering for hooter AK
      O_HooterAS1 { ExternalAccessible := 'False'; ExternalVisible := 'False'; ExternalWritable := 'False'} : Bool;   // Steering for hooter AS1
      O_HooterAS2 { ExternalAccessible := 'False'; ExternalVisible := 'False'; ExternalWritable := 'False'} : Bool;   // Steering for hooter AS2
      O_FlashAK { ExternalAccessible := 'False'; ExternalVisible := 'False'; ExternalWritable := 'False'} : Bool;   // Steering for flashlight AK
      O_FlashAS1 { ExternalAccessible := 'False'; ExternalVisible := 'False'; ExternalWritable := 'False'} : Bool;   // Steering for flashlight AS1
      O_FlashAS2 { ExternalAccessible := 'False'; ExternalVisible := 'False'; ExternalWritable := 'False'} : Bool;   // Steering for flashlight AS2
   END_VAR
   VAR DB_SPECIFIC
      HooterForAlmAB { ExternalAccessible := 'False'; ExternalVisible := 'False'; ExternalWritable := 'False'} : Bool;   // Hooter activation for fault A or B
      HooterForWarnSt { ExternalAccessible := 'False'; ExternalVisible := 'False'; ExternalWritable := 'False'} : Bool;   // Hooter activation for warningstart
      DelayTimeElapsed { ExternalAccessible := 'False'; ExternalVisible := 'False'; ExternalWritable := 'False'} : Bool;   // Timer result (on during max 1 hour)
      ResetDone { ExternalAccessible := 'False'; ExternalVisible := 'False'; ExternalWritable := 'False'} : Bool;   // Reset done
      DelayTimerValue { ExternalAccessible := 'False'; ExternalVisible := 'False'; ExternalWritable := 'False'} : DInt;   // Delay Timer elapsed
   END_VAR
   VAR
      DelayTimer { ExternalAccessible := 'False'; ExternalVisible := 'False'; ExternalWritable := 'False'; S7_SetPoint := 'True'} : "LTimer";
   END_VAR
BEGIN

REGION Network 1: *** 1 - Inputs *** Timer for maximum 1 hour operation of the hooter
   // Timer for maximum 1 hour operation of the hooter
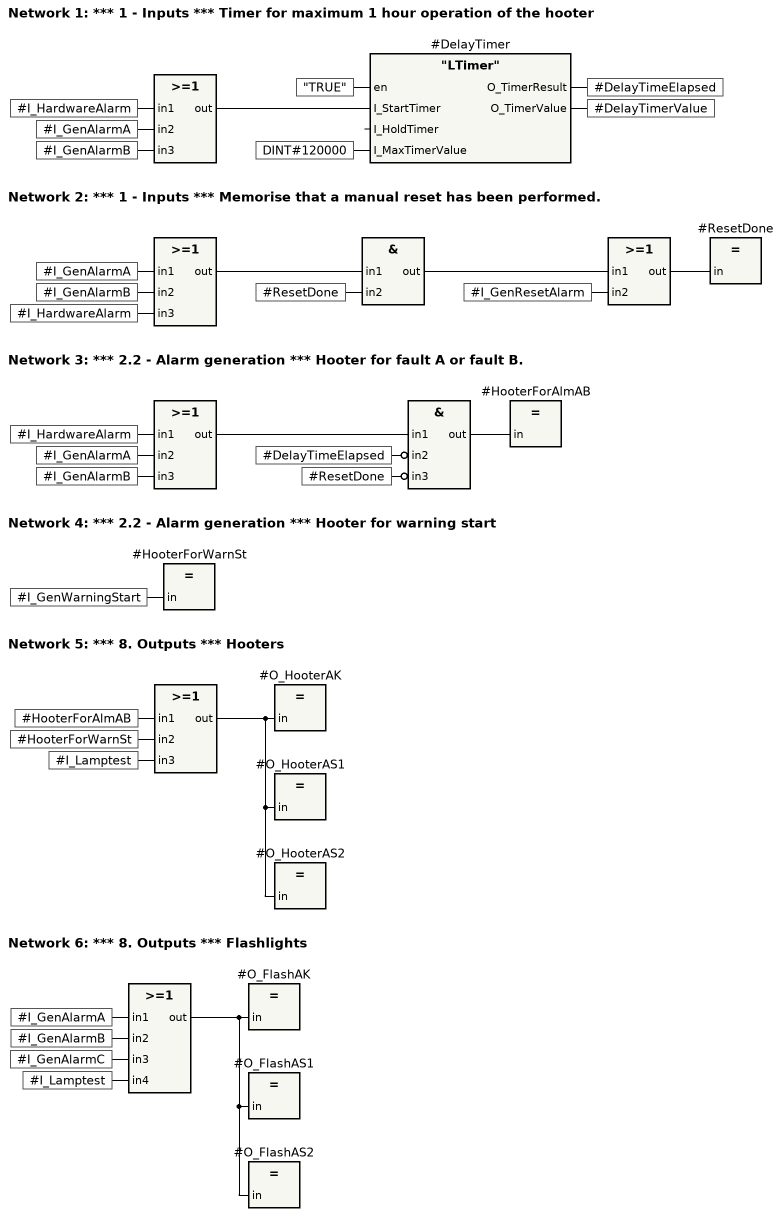
   IF "TRUE" THEN
       #DelayTimer(I_StartTimer := #I_HardwareAlarm OR #I_GenAlarmA OR #I_GenAlarmB,   // "LTimer"
                   I_MaxTimerValue := DINT#120000,
                   O_TimerResult => #DelayTimeElapsed,
                   O_TimerValue => #DelayTimerValue);
   END_IF;
END_REGION

REGION Network 2: *** 1 - Inputs *** Memorise that a manual reset has been performed.
   // Memorise that a manual reset has been performed.
   #ResetDone := ((#I_GenAlarmA OR #I_GenAlarmB OR #I_HardwareAlarm) AND #ResetDone) OR #I_GenResetAlarm;
END_REGION

REGION Network 3: *** 2.2 - Alarm generation *** Hooter for fault A or fault B.
   // Hooter for fault A or fault B.
   // Muted after x time OR when reset button was pressed.
   #HooterForAlmAB := (#I_HardwareAlarm OR #I_GenAlarmA OR #I_GenAlarmB) AND NOT #DelayTimeElapsed AND NOT #ResetDone;
END_REGION

REGION Network 4: *** 2.2 - Alarm generation *** Hooter for warning start
   // Hooter for warning start
   #HooterForWarnSt := #I_GenWarningStart;
END_REGION

REGION Network 5: *** 8. Outputs *** Hooters
   // Hooters
   #O_HooterAK := #HooterForAlmAB OR #HooterForWarnSt OR #I_Lamptest;
   #O_HooterAS1 := #O_HooterAK;
   #O_HooterAS2 := #O_HooterAK;
END_REGION

REGION Network 6: *** 8. Outputs *** Flashlights
   // Flashlights
   #O_FlashAK := #I_GenAlarmA OR #I_GenAlarmB OR #I_GenAlarmC OR #I_Lamptest;
   #O_FlashAS1 := #O_FlashAK;
   #O_FlashAS2 := #O_FlashAK;
END_REGION
END_FUNCTION_BLOCK

FUNCTION_BLOCK "LSafetyCheck"   // FB1008, FBD
TITLE = LSafetyCheck
{ S7_Optimized_Access := 'FALSE' }
AUTHOR : VCC
FAMILY : Control
NAME : SafCheck
VERSION : 1.0
// ================================================================================
// This module controls that the checksum from the failsafe and the hardcoded 
// value in the standard part are the same. It also checks that the failsafe is 
// running.
// ================================================================================
// stored: AutoNumber false, IsIECCheckEnabled false, SetENOAutomatically False, UDAEnableTagReadback false
   VAR_INPUT
      I_FSCheckSum : DWord;   // Failsafe checksum
      I_ConfirmWith : DWord;   // Hardcoded checksum
      I_FailSafeNotRunning { ExternalAccessible := 'False'; ExternalVisible := 'False'; ExternalWritable := 'False'} : Bool;   // Failsafe is not running
      I_AlarmResetPB { ExternalAccessible := 'False'; ExternalVisible := 'False'; ExternalWritable := 'False'} : Bool;   // Alarm reset pushbutton is activated
   END_VAR
   VAR_OUTPUT
      O_AlarmABCondition { ExternalAccessible := 'False'; ExternalVisible := 'False'; ExternalWritable := 'False'} : Bool;   // Alarm AB condition
      O_AlarmA { ExternalAccessible := 'False'; ExternalVisible := 'False'; ExternalWritable := 'False'} : Bool;   // Alarm A
      O_AlarmB { ExternalAccessible := 'False'; ExternalVisible := 'False'; ExternalWritable := 'False'} : Bool;   // Alarm B
      O_AlarmC { ExternalAccessible := 'False'; ExternalVisible := 'False'; ExternalWritable := 'False'} : Bool;   // Alarm C
      O_AlarmD { ExternalAccessible := 'False'; ExternalVisible := 'False'; ExternalWritable := 'False'} : Bool;   // Alarm D
      H_IAnim { ExternalAccessible := 'False'; ExternalVisible := 'False'; ExternalWritable := 'False'} : Word;   // Icon Animation
      H_AlarmWord { ExternalAccessible := 'False'; ExternalVisible := 'False'; ExternalWritable := 'False'} : DWord;   // Alarm Word
   END_VAR
   VAR DB_SPECIFIC
      AA_ChecksumAlarm { ExternalAccessible := 'False'; ExternalVisible := 'False'; ExternalWritable := 'False'} : Bool;   // Wrong checksum in failsafe
      AA_FailsafeNotRunning { ExternalAccessible := 'False'; ExternalVisible := 'False'; ExternalWritable := 'False'} : Bool;   // Failsafe not running
      H_Out : Struct   // HMI
         Anim : Word;   // HMI Animation of the object
         DBnr : Int;   // HMI Animation DB number
      END_STRUCT;
      ChecksumOk { ExternalAccessible := 'False'; ExternalVisible := 'False'; ExternalWritable := 'False'} : Bool := TRUE;   // Checksum is ok
      ChecksumAlarmCond { ExternalAccessible := 'False'; ExternalVisible := 'False'; ExternalWritable := 'False'} : Bool;   // Checksum alarm condition
      FailsafeNotRunningCond { ExternalAccessible := 'False'; ExternalVisible := 'False'; ExternalWritable := 'False'} : Bool;   // Failsafe not running condition
      AlarmA { ExternalAccessible := 'False'; ExternalVisible := 'False'; ExternalWritable := 'False'} : Bool;   // Alarm A active in the FB
      AlarmB { ExternalAccessible := 'False'; ExternalVisible := 'False'; ExternalWritable := 'False'} : Bool;   // Alarm B active in the FB
      AlarmC { ExternalAccessible := 'False'; ExternalVisible := 'False'; ExternalWritable := 'False'} : Bool;   // Alarm C active in the FB
      AlarmD { ExternalAccessible := 'False'; ExternalVisible := 'False'; ExternalWritable := 'False'} : Bool;   // Alarm D active in the FB
      DBNumber { ExternalAccessible := 'False'; ExternalVisible := 'False'; ExternalWritable := 'False'} : Int;   // DB number
      FSCheckSum { ExternalAccessible := 'False'; ExternalVisible := 'False'; ExternalWritable := 'False'} : DInt;   // Failsafe checksum
      ConfirmWith { ExternalAccessible := 'False'; ExternalVisible := 'False'; ExternalWritable := 'False'} : DInt;   // Hardcoded checksum
      DBnr { ExternalAccessible := 'False'; ExternalVisible := 'False'; ExternalWritable := 'False'} : Int;   // HMI DB number
   END_VAR
BEGIN

NETWORK
TITLE = **** 1 - Inputs **** DB number
// DB number
      L     DINO;
      T     #DBnr;

REGION Network 2: **** 1 - Inputs **** Convert DWORD to DINT
   // Convert DWORD to DINT
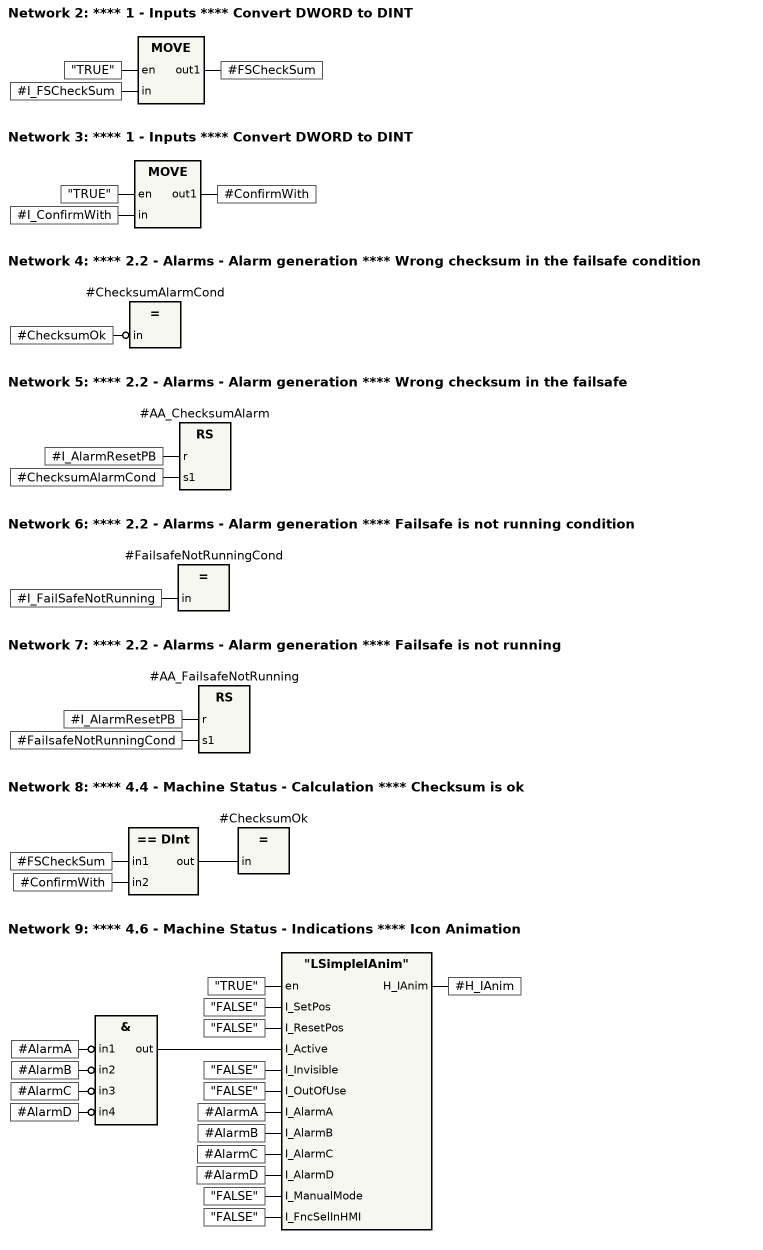
   IF "TRUE" THEN #FSCheckSum := #I_FSCheckSum; END_IF;
END_REGION

REGION Network 3: **** 1 - Inputs **** Convert DWORD to DINT
   // Convert DWORD to DINT
   IF "TRUE" THEN #ConfirmWith := #I_ConfirmWith; END_IF;
END_REGION

REGION Network 4: **** 2.2 - Alarms - Alarm generation **** Wrong checksum in the failsafe condition
   // Wrong checksum in the failsafe condition
   #ChecksumAlarmCond := NOT #ChecksumOk;
END_REGION

REGION Network 5: **** 2.2 - Alarms - Alarm generation **** Wrong checksum in the failsafe
   // Wrong checksum in the failsafe
   IF #I_AlarmResetPB THEN
       #AA_ChecksumAlarm := FALSE;   // RS flip-flop
   END_IF;
   IF #ChecksumAlarmCond THEN #AA_ChecksumAlarm := TRUE; END_IF;
END_REGION

REGION Network 6: **** 2.2 - Alarms - Alarm generation **** Failsafe is not running condition
   // Failsafe is not running condition
   #FailsafeNotRunningCond := #I_FailSafeNotRunning;
END_REGION

REGION Network 7: **** 2.2 - Alarms - Alarm generation **** Failsafe is not running
   // Failsafe is not running
   IF #I_AlarmResetPB THEN
       #AA_FailsafeNotRunning := FALSE;   // RS flip-flop
   END_IF;
   IF #FailsafeNotRunningCond THEN #AA_FailsafeNotRunning := TRUE; END_IF;
END_REGION

REGION Network 8: **** 4.4 - Machine Status - Calculation **** Checksum is ok
   // Checksum is ok
   #ChecksumOk := #FSCheckSum = #ConfirmWith;
END_REGION

REGION Network 9: **** 4.6 - Machine Status - Indications **** Icon Animation
   // Icon Animation
   IF "TRUE" THEN
       "LSimpleIAnim"(I_SetPos := "FALSE",
                      I_ResetPos := "FALSE",
                      I_Active := NOT #AlarmA AND NOT #AlarmB AND NOT #AlarmC AND NOT #AlarmD,
                      I_Invisible := "FALSE",
                      I_OutOfUse := "FALSE",
                      I_AlarmA := #AlarmA,
                      I_AlarmB := #AlarmB,
                      I_AlarmC := #AlarmC,
                      I_AlarmD := #AlarmD,
                      I_ManualMode := "FALSE",
                      I_FncSelInHMI := "FALSE",
                      H_IAnim => #H_IAnim);
   END_IF;
END_REGION

REGION Network 10: **** 4.6 - Machine Status - Indications **** Animation
   // Animation
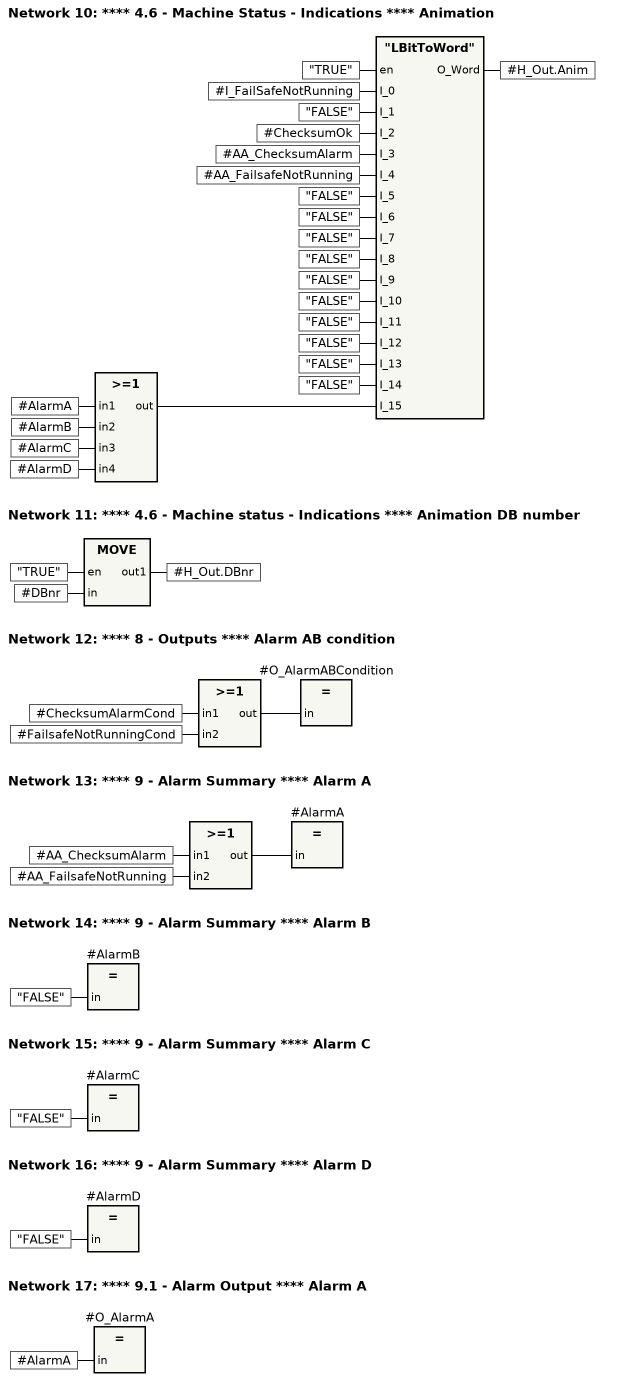
   IF "TRUE" THEN
       "LBitToWord"(I_0 := #I_FailSafeNotRunning,
                    I_1 := "FALSE",
                    I_2 := #ChecksumOk,
                    I_3 := #AA_ChecksumAlarm,
                    I_4 := #AA_FailsafeNotRunning,
                    I_5 := "FALSE",
                    I_6 := "FALSE",
                    I_7 := "FALSE",
                    I_8 := "FALSE",
                    I_9 := "FALSE",
                    I_10 := "FALSE",
                    I_11 := "FALSE",
                    I_12 := "FALSE",
                    I_13 := "FALSE",
                    I_14 := "FALSE",
                    I_15 := #AlarmA OR #AlarmB OR #AlarmC OR #AlarmD,
                    O_Word => #H_Out.Anim);
   END_IF;
END_REGION

REGION Network 11: **** 4.6 - Machine status - Indications **** Animation DB number
   // Animation DB number
   IF "TRUE" THEN #H_Out.DBnr := #DBnr; END_IF;
END_REGION

REGION Network 12: **** 8 - Outputs **** Alarm AB condition
   // Alarm AB condition
   #O_AlarmABCondition := #ChecksumAlarmCond OR #FailsafeNotRunningCond;
END_REGION

REGION Network 13: **** 9 - Alarm Summary **** Alarm A
   // Summary of alarms A
   #AlarmA := #AA_ChecksumAlarm OR #AA_FailsafeNotRunning;
END_REGION

REGION Network 14: **** 9 - Alarm Summary **** Alarm B
   // Summary of alarms B
   #AlarmB := "FALSE";
END_REGION

REGION Network 15: **** 9 - Alarm Summary **** Alarm C
   // Summary of alarms C
   #AlarmC := "FALSE";
END_REGION

REGION Network 16: **** 9 - Alarm Summary **** Alarm D
   // Summary of alarms D
   #AlarmD := "FALSE";
END_REGION

REGION Network 17: **** 9.1 - Alarm Output **** Alarm A
   // Summary of alarms A
   #O_AlarmA := #AlarmA;
END_REGION

REGION Network 18: **** 9.1 - Alarm Output **** Alarm B
   // Summary of alarms B
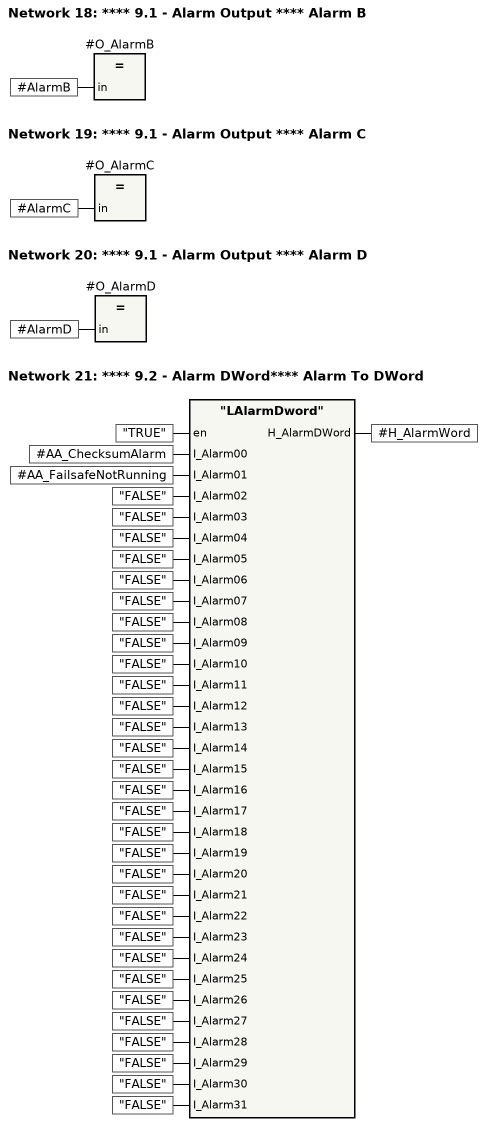
   #O_AlarmB := #AlarmB;
END_REGION

REGION Network 19: **** 9.1 - Alarm Output **** Alarm C
   // Summary of alarms C
   #O_AlarmC := #AlarmC;
END_REGION

REGION Network 20: **** 9.1 - Alarm Output **** Alarm D
   // Summary of alarms D
   #O_AlarmD := #AlarmD;
END_REGION

REGION Network 21: **** 9.2 - Alarm DWord**** Alarm To DWord
   // Alarm Word
   IF "TRUE" THEN
       "LAlarmDword"(I_Alarm00 := #AA_ChecksumAlarm,
                     I_Alarm01 := #AA_FailsafeNotRunning,
                     I_Alarm02 := "FALSE",
                     I_Alarm03 := "FALSE",
                     I_Alarm04 := "FALSE",
                     I_Alarm05 := "FALSE",
                     I_Alarm06 := "FALSE",
                     I_Alarm07 := "FALSE",
                     I_Alarm08 := "FALSE",
                     I_Alarm09 := "FALSE",
                     I_Alarm10 := "FALSE",
                     I_Alarm11 := "FALSE",
                     I_Alarm12 := "FALSE",
                     I_Alarm13 := "FALSE",
                     I_Alarm14 := "FALSE",
                     I_Alarm15 := "FALSE",
                     I_Alarm16 := "FALSE",
                     I_Alarm17 := "FALSE",
                     I_Alarm18 := "FALSE",
                     I_Alarm19 := "FALSE",
                     I_Alarm20 := "FALSE",
                     I_Alarm21 := "FALSE",
                     I_Alarm22 := "FALSE",
                     I_Alarm23 := "FALSE",
                     I_Alarm24 := "FALSE",
                     I_Alarm25 := "FALSE",
                     I_Alarm26 := "FALSE",
                     I_Alarm27 := "FALSE",
                     I_Alarm28 := "FALSE",
                     I_Alarm29 := "FALSE",
                     I_Alarm30 := "FALSE",
                     I_Alarm31 := "FALSE",
                     H_AlarmDWord => #H_AlarmWord);
   END_IF;
END_REGION
END_FUNCTION_BLOCK

FUNCTION_BLOCK "LPulsesGenerator"   // FB1010, FBD
TITLE = LPulsesGenerator
{ S7_Optimized_Access := 'FALSE' }
AUTHOR : VCC
FAMILY : Control
NAME : PulseGen
VERSION : 1.0
// ================================================================================
// LPulsesGenerator is used everywhere a pulse signal is requiered.
// This function is able to generate pulse without disturbance due to scan time of 
// CPU. This function is able to generate pulse with a fix frequency.
// This function is also able to generate pulse with a defined time ON and a 
// different Time OFF.
// It is also possible to hold the function.
// It is also possible to use the running value of time ON and time OFF.
// ================================================================================
// stored: AutoNumber false, IsIECCheckEnabled false, SetENOAutomatically False, UDAEnableTagReadback false
   VAR_INPUT
      I_Input { ExternalAccessible := 'False'; ExternalVisible := 'False'; ExternalWritable := 'False'} : Bool;   // Input to start pulse generator
      I_Hold { ExternalAccessible := 'False'; ExternalVisible := 'False'; ExternalWritable := 'False'} : Bool;   // Input to hold the pulse generator
      I_Frequency { ExternalAccessible := 'False'; ExternalVisible := 'False'; ExternalWritable := 'False'} : DInt;   // Input to generated pulses to this frequency
      I_TimeOFF { ExternalAccessible := 'False'; ExternalVisible := 'False'; ExternalWritable := 'False'} : DInt;   // Duration OFF for pulses
      I_TimeON { ExternalAccessible := 'False'; ExternalVisible := 'False'; ExternalWritable := 'False'} : DInt;   // Duration ON for pulses
   END_VAR
   VAR_OUTPUT
      O_Pulses { ExternalAccessible := 'False'; ExternalVisible := 'False'; ExternalWritable := 'False'} : Bool;   // Pulses
      O_TimeOFF { ExternalAccessible := 'False'; ExternalVisible := 'False'; ExternalWritable := 'False'} : DInt;   // Value TimerOFF period
      O_TimeON { ExternalAccessible := 'False'; ExternalVisible := 'False'; ExternalWritable := 'False'} : DInt;   // Value TimerON period
   END_VAR
   VAR DB_SPECIFIC
      OFF_Finished { ExternalAccessible := 'False'; ExternalVisible := 'False'; ExternalWritable := 'False'} : Bool;   // Signal when timer OFF period finished
      ON_Finished { ExternalAccessible := 'False'; ExternalVisible := 'False'; ExternalWritable := 'False'} : Bool;   // Signal when timer ON period finished
      TimeOFF { ExternalAccessible := 'False'; ExternalVisible := 'False'; ExternalWritable := 'False'} : DInt;   // Duration OFF for pulses
      TimeON { ExternalAccessible := 'False'; ExternalVisible := 'False'; ExternalWritable := 'False'} : DInt;   // Duration ON for pulses
      OFF_FinishPulse { ExternalAccessible := 'False'; ExternalVisible := 'False'; ExternalWritable := 'False'} : Bool;   // Off Finished pulse
      RunningTimeOFF { ExternalAccessible := 'False'; ExternalVisible := 'False'; ExternalWritable := 'False'} : DInt;   // Duration OFF for pulses
      TimeOffOT { ExternalAccessible := 'False'; ExternalVisible := 'False'; ExternalWritable := 'False'} : DInt;   // Overtime for timer off
      TimeOffOTAcc { ExternalAccessible := 'False'; ExternalVisible := 'False'; ExternalWritable := 'False'} : DInt;   // Acculumated overtime for timer off
      TimeOffAdj { ExternalAccessible := 'False'; ExternalVisible := 'False'; ExternalWritable := 'False'} : DInt;   // Adjusted value for Timer off
      ON_FinishPulse { ExternalAccessible := 'False'; ExternalVisible := 'False'; ExternalWritable := 'False'} : Bool;   // On Finished pulse
      RunningTimeON { ExternalAccessible := 'False'; ExternalVisible := 'False'; ExternalWritable := 'False'} : DInt;   // Duration OFF for pulses
      TimeOnOT { ExternalAccessible := 'False'; ExternalVisible := 'False'; ExternalWritable := 'False'} : DInt;   // Overtime for timer on
      TimeOnOTAcc { ExternalAccessible := 'False'; ExternalVisible := 'False'; ExternalWritable := 'False'} : DInt;   // Acculumated overtime for timer on
      TimeOnAdj { ExternalAccessible := 'False'; ExternalVisible := 'False'; ExternalWritable := 'False'} : DInt;   // Adjusted value for Timer on
   END_VAR
   VAR
      TimerOFFPer { ExternalAccessible := 'False'; ExternalVisible := 'False'; ExternalWritable := 'False'; S7_SetPoint := 'True'} : "LTimer";   // Timer OFF period
      TimerONPer { ExternalAccessible := 'False'; ExternalVisible := 'False'; ExternalWritable := 'False'; S7_SetPoint := 'True'} : "LTimer";   // Timer ON period
   END_VAR
   VAR_TEMP
      Frequency : DInt;   // Temp frequency
   END_VAR
   VAR_TEMP   // added for the SCL form of the ladder/FBD networks
      _w1 : Bool;
      _w2 : Bool;
   END_VAR
BEGIN

REGION Network 1: **** 4.4 - Machine Status - Calculated **** Reset all timer values
   // Reset all timer values
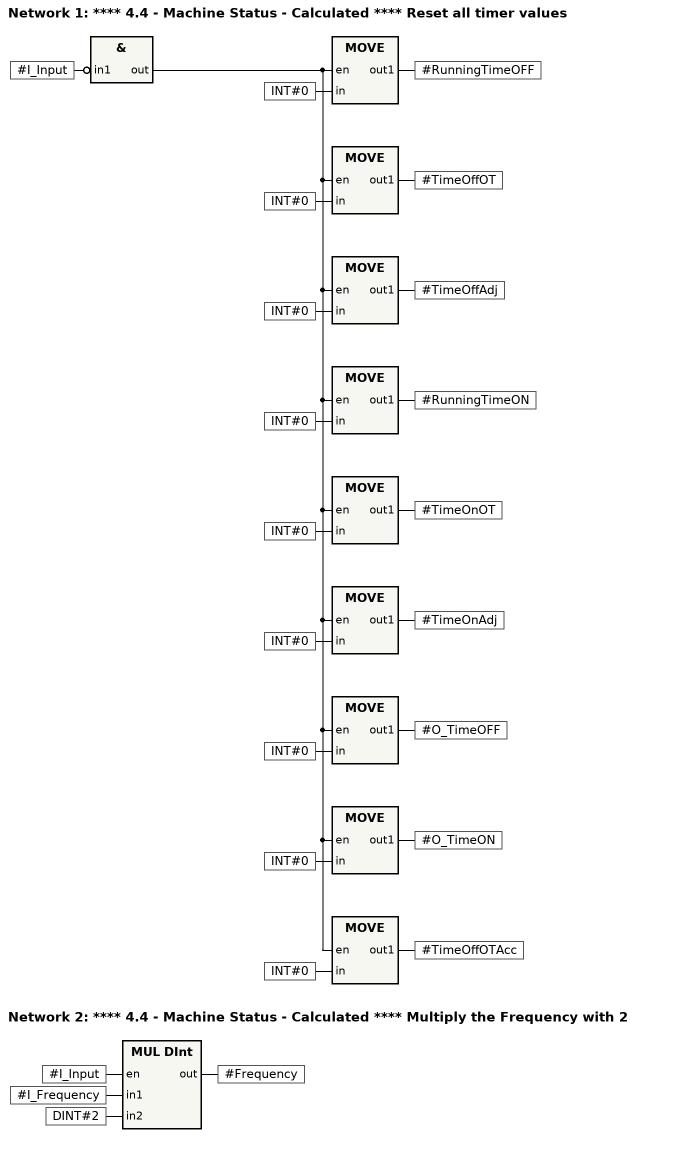
   IF NOT #I_Input THEN
       #RunningTimeOFF := INT#0;
       #TimeOffOT := INT#0;
       #TimeOffAdj := INT#0;
       #RunningTimeON := INT#0;
       #TimeOnOT := INT#0;
       #TimeOnAdj := INT#0;
       #O_TimeOFF := INT#0;
       #O_TimeON := INT#0;
       #TimeOffOTAcc := INT#0;
   END_IF;
END_REGION

REGION Network 2: **** 4.4 - Machine Status - Calculated **** Multiply the Frequency with 2
   // Multiply the Frequency with 2
   IF #I_Input THEN #Frequency := #I_Frequency * DINT#2; END_IF;
END_REGION

REGION Network 3: **** 4.4 - Machine Status - Calculated **** Calculation of TimeOFF and TimeON if I_Frequemcy selected
   // Calculation of TimeOFF and TimeON if I_Frequemcy selected
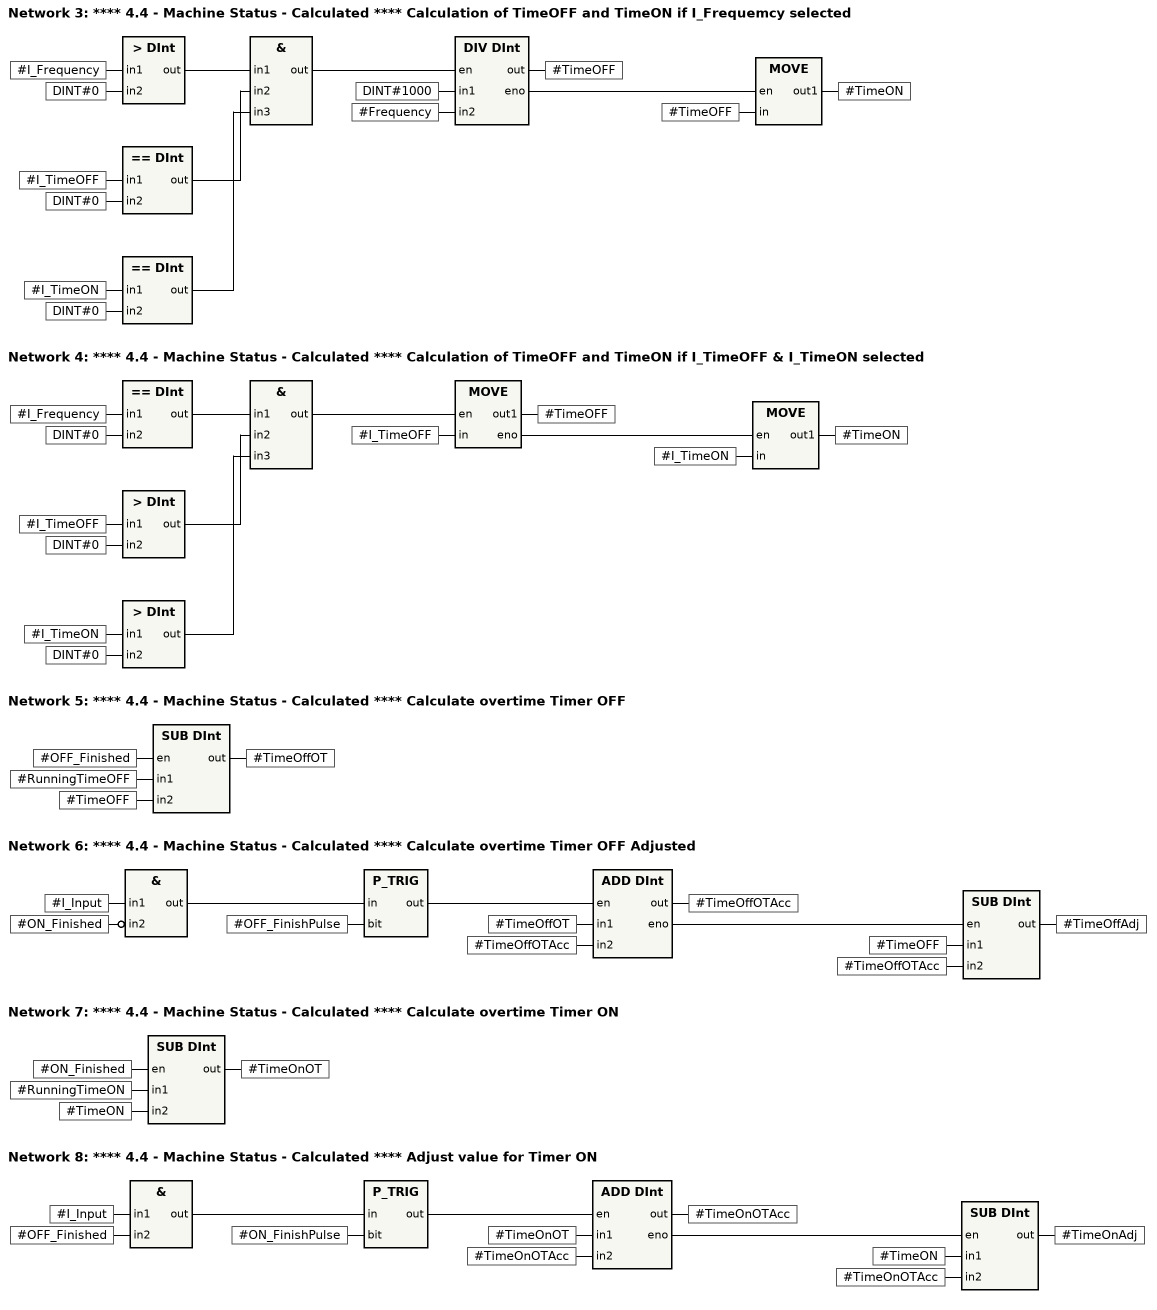
   // ENO of a box is taken as its EN; it also drops when the box reports an error
   IF (#I_Frequency > DINT#0) AND (#I_TimeOFF = DINT#0) AND (#I_TimeON = DINT#0) THEN
       #TimeOFF := DINT#1000 / #Frequency;
       #TimeON := #TimeOFF;
   END_IF;
END_REGION

REGION Network 4: **** 4.4 - Machine Status - Calculated **** Calculation of TimeOFF and TimeON if I_TimeOFF & I_TimeON selected
   // Calculation of TimeOFF and TimeON if I_TimeOFF & I_TimeON selected
   // ENO of a box is taken as its EN; it also drops when the box reports an error
   IF (#I_Frequency = DINT#0) AND (#I_TimeOFF > DINT#0) AND (#I_TimeON > DINT#0) THEN
       #TimeOFF := #I_TimeOFF;
       #TimeON := #I_TimeON;
   END_IF;
END_REGION

REGION Network 5: **** 4.4 - Machine Status - Calculated **** Calculate overtime Timer OFF
   // Calculate overtime Timer OFF
   IF #OFF_Finished THEN #TimeOffOT := #RunningTimeOFF - #TimeOFF; END_IF;
END_REGION

REGION Network 6: **** 4.4 - Machine Status - Calculated **** Calculate overtime Timer OFF Adjusted
   // Calculate overtime Timer OFF Adjusted
   // ENO of a box is taken as its EN; it also drops when the box reports an error
   #_w1 := #I_Input AND NOT #ON_Finished;
   #_w2 := #_w1 AND NOT #OFF_FinishPulse;   // rising edge
   #OFF_FinishPulse := #_w1;
   IF #_w2 THEN
       #TimeOffOTAcc := #TimeOffOT + #TimeOffOTAcc;
       #TimeOffAdj := #TimeOFF - #TimeOffOTAcc;
   END_IF;
END_REGION

REGION Network 7: **** 4.4 - Machine Status - Calculated **** Calculate overtime Timer ON
   // Calculate overtime Timer ON
   IF #ON_Finished THEN #TimeOnOT := #RunningTimeON - #TimeON; END_IF;
END_REGION

REGION Network 8: **** 4.4 - Machine Status - Calculated **** Adjust value for Timer ON
   // Adjust value for Timer ON
   // ENO of a box is taken as its EN; it also drops when the box reports an error
   #_w1 := #I_Input AND #OFF_Finished;
   #_w2 := #_w1 AND NOT #ON_FinishPulse;   // rising edge
   #ON_FinishPulse := #_w1;
   IF #_w2 THEN
       #TimeOnOTAcc := #TimeOnOT + #TimeOnOTAcc;
       #TimeOnAdj := #TimeON - #TimeOnOTAcc;
   END_IF;
END_REGION

REGION Network 9: **** 4.4 - Machine Status - Calculated **** Timer to generated Time OFF
   // Timer to generated Time OFF
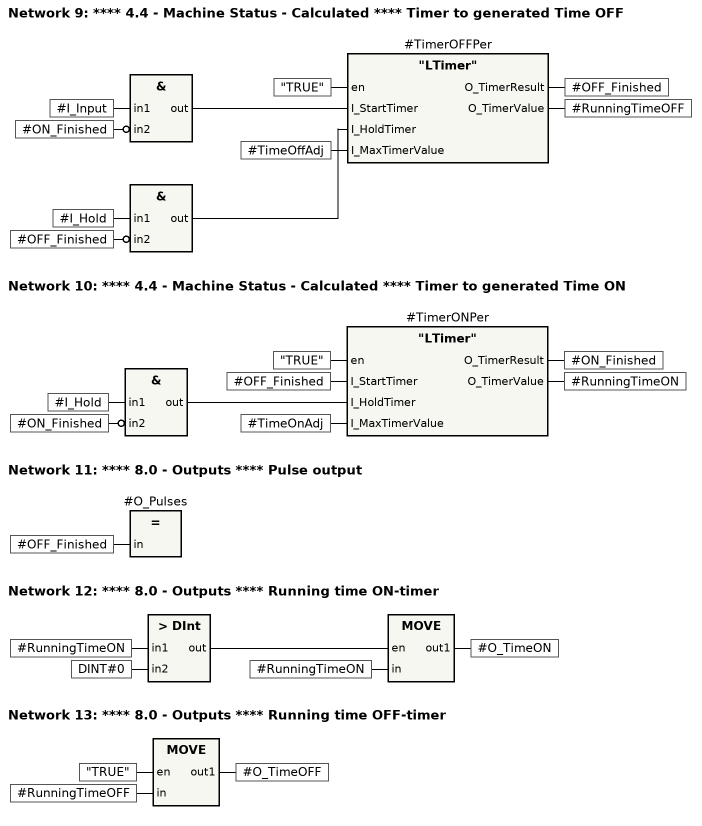
   IF "TRUE" THEN
       #TimerOFFPer(I_StartTimer := #I_Input AND NOT #ON_Finished,   // "LTimer"
                    I_HoldTimer := #I_Hold AND NOT #OFF_Finished,
                    I_MaxTimerValue := #TimeOffAdj,
                    O_TimerResult => #OFF_Finished,
                    O_TimerValue => #RunningTimeOFF);
   END_IF;
END_REGION

REGION Network 10: **** 4.4 - Machine Status - Calculated **** Timer to generated Time ON
   // Timer to generated Time ON
   IF "TRUE" THEN
       #TimerONPer(I_StartTimer := #OFF_Finished,   // "LTimer"
                   I_HoldTimer := #I_Hold AND NOT #ON_Finished,
                   I_MaxTimerValue := #TimeOnAdj,
                   O_TimerResult => #ON_Finished,
                   O_TimerValue => #RunningTimeON);
   END_IF;
END_REGION

REGION Network 11: **** 8.0 - Outputs **** Pulse output
   // Pulse output
   #O_Pulses := #OFF_Finished;
END_REGION

REGION Network 12: **** 8.0 - Outputs **** Running time ON-timer
   // Running time ON-timer
   IF #RunningTimeON > DINT#0 THEN #O_TimeON := #RunningTimeON; END_IF;
END_REGION

REGION Network 13: **** 8.0 - Outputs **** Running time OFF-timer
   // Running time OFF-timer
   IF "TRUE" THEN #O_TimeOFF := #RunningTimeOFF; END_IF;
END_REGION
END_FUNCTION_BLOCK

FUNCTION_BLOCK "LPulse"   // FB1013, FBD
TITLE = LPulse
{ S7_Optimized_Access := 'FALSE' }
AUTHOR : VCC
FAMILY : Control
NAME : TimerON
VERSION : 1.0
// ================================================================================
// LPulse is used when a delay is necessary without using timer from Siemens.
// This timer has 2 ways to run:
// * Input = true constantly and pulse output 
// 
// Timer reset when input = false
// Timer reset when input reset = true 
// 
// For each case, Timer is reset when O_TimerValue >= I_MaxTimerValue
// ================================================================================
// stored: AutoNumber false, IsIECCheckEnabled false, SetENOAutomatically False, UDAEnableTagReadback false
   VAR_INPUT
      I_StartTimer { ExternalAccessible := 'False'; ExternalVisible := 'False'; ExternalWritable := 'False'} : Bool;   // Start Timer
      I_ResetTimer { ExternalAccessible := 'False'; ExternalVisible := 'False'; ExternalWritable := 'False'} : Bool;   // ResetTimer when I_MemstartTimer active
      I_MaxTimerValue { ExternalAccessible := 'False'; ExternalVisible := 'False'; ExternalWritable := 'False'} : DInt;   // Maximum Timer Value (1 unit = 1ms and max=7FFFFFFF)
   END_VAR
   VAR_OUTPUT
      O_TimerResult { ExternalAccessible := 'False'; ExternalVisible := 'False'; ExternalWritable := 'False'} : Bool;   // Timer result when time = MaxTime
      O_TimerValue { ExternalAccessible := 'False'; ExternalVisible := 'False'; ExternalWritable := 'False'} : DInt;   // Current timer value
   END_VAR
   VAR DB_SPECIFIC
      PulseStart { ExternalAccessible := 'False'; ExternalVisible := 'False'; ExternalWritable := 'False'} : Bool;   // Positive Pulse Start Timer
      MemStartTimer { ExternalAccessible := 'False'; ExternalVisible := 'False'; ExternalWritable := 'False'} : Bool;   // Memory of start timer
      PulseMemStart { ExternalAccessible := 'False'; ExternalVisible := 'False'; ExternalWritable := 'False'} : Bool;   // Positive Pulse Memory Start Timer
      StartTimeValue { ExternalAccessible := 'False'; ExternalVisible := 'False'; ExternalWritable := 'False'} : DInt;   // Start time value
      RunningTimeValue { ExternalAccessible := 'False'; ExternalVisible := 'False'; ExternalWritable := 'False'} : DInt;   // Running time value
      ElapsedTimeValue { ExternalAccessible := 'False'; ExternalVisible := 'False'; ExternalWritable := 'False'} : DInt;   // elapsed time value
   END_VAR
   VAR_TEMP
      T_Int : DInt;   // Temporally value
   END_VAR
   VAR_TEMP   // added for the SCL form of the ladder/FBD networks
      _w1 : Bool;
   END_VAR
BEGIN

REGION Network 1: **** 4.4 - Machine Status - Calculated **** Timer is running
   // Timer is running
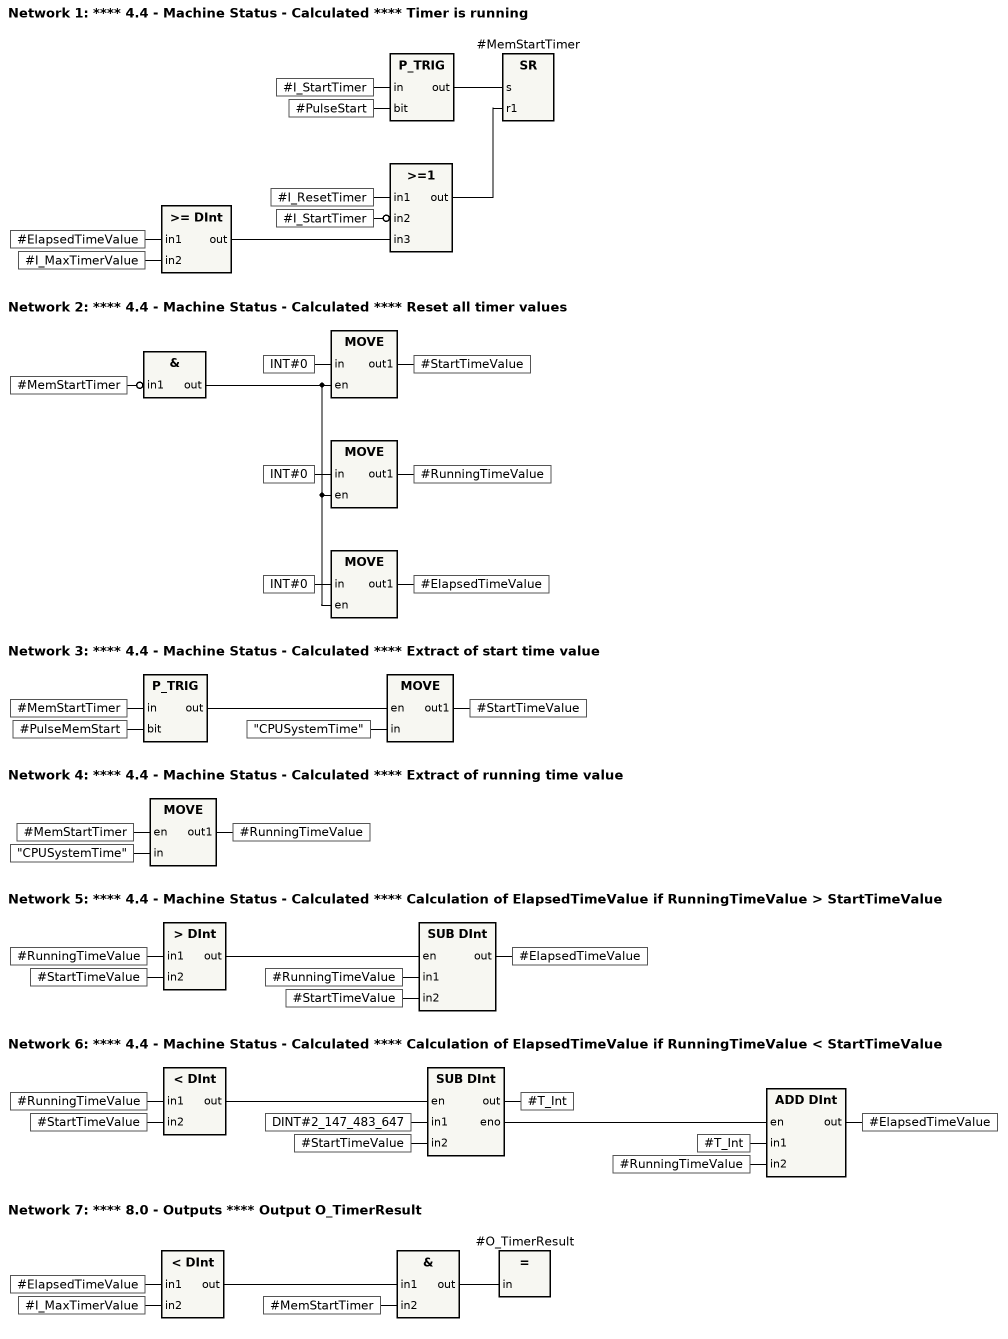
   #_w1 := #I_StartTimer AND NOT #PulseStart;   // rising edge
   #PulseStart := #I_StartTimer;
   IF #_w1 THEN
       #MemStartTimer := TRUE;   // SR flip-flop
   END_IF;
   IF #I_ResetTimer OR NOT #I_StartTimer OR (#ElapsedTimeValue >= #I_MaxTimerValue) THEN
       #MemStartTimer := FALSE;
   END_IF;
END_REGION

REGION Network 2: **** 4.4 - Machine Status - Calculated **** Reset all timer values
   // Reset all timer values
   IF NOT #MemStartTimer THEN
       #StartTimeValue := INT#0;
       #RunningTimeValue := INT#0;
       #ElapsedTimeValue := INT#0;
   END_IF;
END_REGION

REGION Network 3: **** 4.4 - Machine Status - Calculated **** Extract of start time value
   // Extract of start time value
   #_w1 := #MemStartTimer AND NOT #PulseMemStart;   // rising edge
   #PulseMemStart := #MemStartTimer;
   IF #_w1 THEN #StartTimeValue := "CPUSystemTime"; END_IF;
END_REGION

REGION Network 4: **** 4.4 - Machine Status - Calculated **** Extract of running time value
   // Extract of running time value
   IF #MemStartTimer THEN #RunningTimeValue := "CPUSystemTime"; END_IF;
END_REGION

REGION Network 5: **** 4.4 - Machine Status - Calculated **** Calculation of ElapsedTimeValue if RunningTimeValue > StartTimeValue
   // Calculation of ElapsedTimeValue if RunningTimeValue > StartTimeValue
   IF #RunningTimeValue > #StartTimeValue THEN
       #ElapsedTimeValue := #RunningTimeValue - #StartTimeValue;
   END_IF;
END_REGION

REGION Network 6: **** 4.4 - Machine Status - Calculated **** Calculation of ElapsedTimeValue if RunningTimeValue < StartTimeValue
   // Calculation of ElapsedTimeValue if RunningTimeValue < StartTimeValue
   // ENO of a box is taken as its EN; it also drops when the box reports an error
   IF #RunningTimeValue < #StartTimeValue THEN
       #T_Int := DINT#2_147_483_647 - #StartTimeValue;
       #ElapsedTimeValue := #T_Int + #RunningTimeValue;
   END_IF;
END_REGION

REGION Network 7: **** 8.0 - Outputs **** Output O_TimerResult
   // Output O_TimerResult
   #O_TimerResult := (#ElapsedTimeValue < #I_MaxTimerValue) AND #MemStartTimer;
END_REGION

REGION Network 8: **** 8.0 - Outputs **** Copy of TimerValue to output O_TimerValue
   // Copy of TimerValue to output O_TimerValue
   // Copy of HoldValue to output O_HoldValue
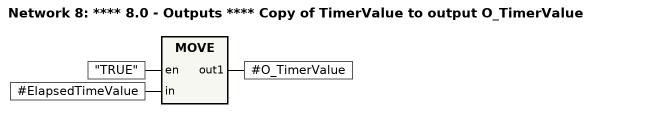
   IF "TRUE" THEN #O_TimerValue := #ElapsedTimeValue; END_IF;
END_REGION
END_FUNCTION_BLOCK

FUNCTION_BLOCK "LConditionDelay"   // FB1101, FBD
TITLE = LConditionDelay
{ S7_Optimized_Access := 'FALSE' }
VERSION : 0.1
// stored: AutoNumber false, IsIECCheckEnabled false, SetENOAutomatically False, UDAEnableTagReadback false
   VAR_INPUT
      I_Condition { ExternalAccessible := 'False'; ExternalVisible := 'False'; ExternalWritable := 'False'} : Bool;   // Condition
      I_ExtDelayTime { ExternalAccessible := 'False'; ExternalVisible := 'False'; ExternalWritable := 'False'} : DInt;   // External delay time
      I_ActivedExtDelayTime { ExternalAccessible := 'False'; ExternalVisible := 'False'; ExternalWritable := 'False'} : Bool;   // Activated external delay time
      I_HoldCond { ExternalAccessible := 'False'; ExternalVisible := 'False'; ExternalWritable := 'False'} : Bool;   // Hold condition normal open
      I_ResetCond { ExternalAccessible := 'False'; ExternalVisible := 'False'; ExternalWritable := 'False'} : Bool;   // Reset condition normal open
      I_BypassCond { ExternalAccessible := 'False'; ExternalVisible := 'False'; ExternalWritable := 'False'} : Bool;   // Bypass condition normal open
   END_VAR
   VAR_OUTPUT
      O_ConditionDelayed { ExternalAccessible := 'False'; ExternalVisible := 'False'; ExternalWritable := 'False'} : Bool;   // Condition delayed
   END_VAR
   VAR_IN_OUT
      H_HMI : "H_HMI";   // Animation
      H_ConditionDelay : "H_ConditionDelay";   // Animation
   END_VAR
   VAR DB_SPECIFIC
      TimerResult { ExternalAccessible := 'False'; ExternalVisible := 'False'; ExternalWritable := 'False'} : Bool;   // Timer result
      TimerValue { ExternalAccessible := 'False'; ExternalVisible := 'False'; ExternalWritable := 'False'} : DInt;   // Timer value
      TimerValueElapsed { ExternalAccessible := 'False'; ExternalVisible := 'False'; ExternalWritable := 'False'} : DInt;   // Timer value elapsed
      TimerExtValue { ExternalAccessible := 'False'; ExternalVisible := 'False'; ExternalWritable := 'False'} : DInt;   // Timer external value
      PrevExtDelayTime { ExternalAccessible := 'False'; ExternalVisible := 'False'; ExternalWritable := 'False'} : DInt;   // Previous external delay time
   END_VAR
   VAR
      DelayTimer { ExternalAccessible := 'False'; ExternalVisible := 'False'; ExternalWritable := 'False'} : "LTimer";   // Timer
   END_VAR
   VAR DB_SPECIFIC
      Edge { ExternalAccessible := 'False'; ExternalVisible := 'False'; ExternalWritable := 'False'} : Array[1..10] of Bool;   // Edge
   END_VAR
   VAR_TEMP   // added for the SCL form of the ladder/FBD networks
      _w1 : Bool;
      _w2 : Bool;
   END_VAR
BEGIN

REGION Network 1: **** 5.2 - Equations **** Timer External Value
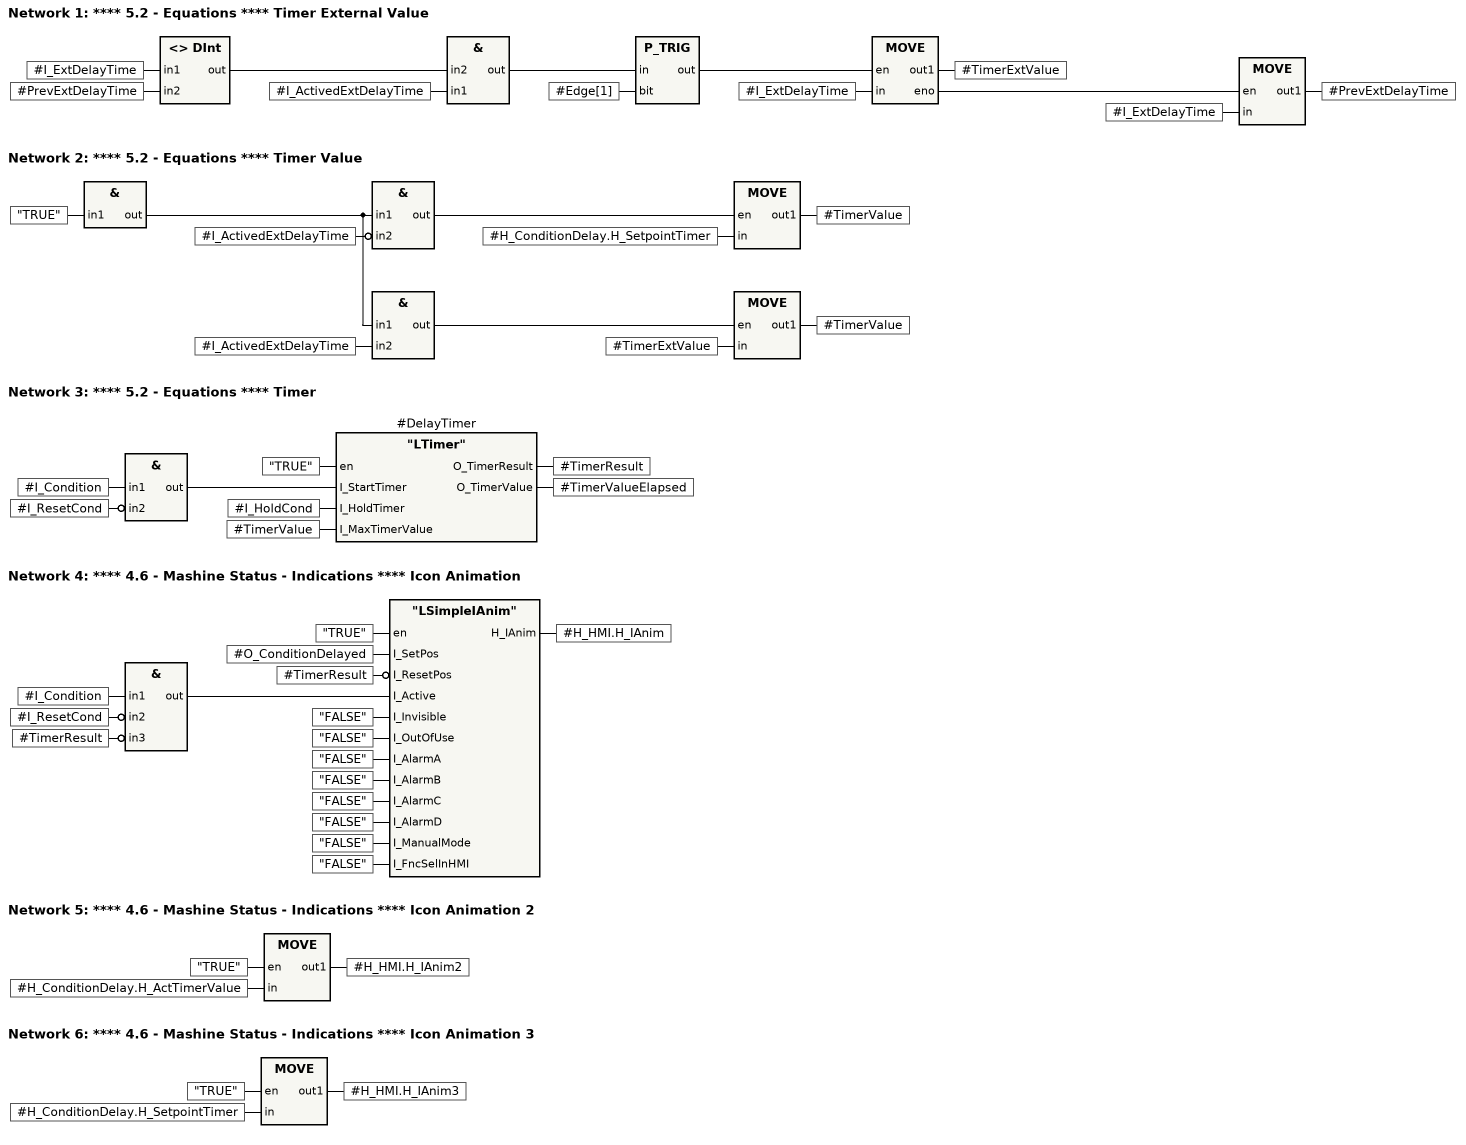
   #_w1 := (#I_ExtDelayTime <> #PrevExtDelayTime) AND #I_ActivedExtDelayTime;
   #_w2 := #_w1 AND NOT #Edge[1];   // rising edge
   #Edge[1] := #_w1;
   IF #_w2 THEN
       #TimerExtValue := #I_ExtDelayTime;
       #PrevExtDelayTime := #I_ExtDelayTime;
   END_IF;
END_REGION

REGION Network 2: **** 5.2 - Equations **** Timer Value
   IF "TRUE" AND NOT #I_ActivedExtDelayTime THEN #TimerValue := #H_ConditionDelay.H_SetpointTimer; END_IF;
   IF "TRUE" AND #I_ActivedExtDelayTime THEN #TimerValue := #TimerExtValue; END_IF;
END_REGION

REGION Network 3: **** 5.2 - Equations **** Timer
   IF "TRUE" THEN
       #DelayTimer(I_StartTimer := #I_Condition AND NOT #I_ResetCond,   // "LTimer"
                   I_HoldTimer := #I_HoldCond,
                   I_MaxTimerValue := #TimerValue,
                   O_TimerResult => #TimerResult,
                   O_TimerValue => #TimerValueElapsed);
   END_IF;
END_REGION

REGION Network 4: **** 4.6 - Mashine Status - Indications **** Icon Animation
   // Icon Animation
   IF "TRUE" THEN
       "LSimpleIAnim"(I_SetPos := #O_ConditionDelayed,
                      I_ResetPos := NOT #TimerResult,
                      I_Active := #I_Condition AND NOT #I_ResetCond AND NOT #TimerResult,
                      I_Invisible := "FALSE",
                      I_OutOfUse := "FALSE",
                      I_AlarmA := "FALSE",
                      I_AlarmB := "FALSE",
                      I_AlarmC := "FALSE",
                      I_AlarmD := "FALSE",
                      I_ManualMode := "FALSE",
                      I_FncSelInHMI := "FALSE",
                      H_IAnim => #H_HMI.H_IAnim);
   END_IF;
END_REGION

REGION Network 5: **** 4.6 - Mashine Status - Indications **** Icon Animation 2
   IF "TRUE" THEN #H_HMI.H_IAnim2 := #H_ConditionDelay.H_ActTimerValue; END_IF;
END_REGION

REGION Network 6: **** 4.6 - Mashine Status - Indications **** Icon Animation 3
   IF "TRUE" THEN #H_HMI.H_IAnim3 := #H_ConditionDelay.H_SetpointTimer; END_IF;
END_REGION

REGION Network 7: **** 4.6 - Machine Status - Indications **** Animation
   // Animation
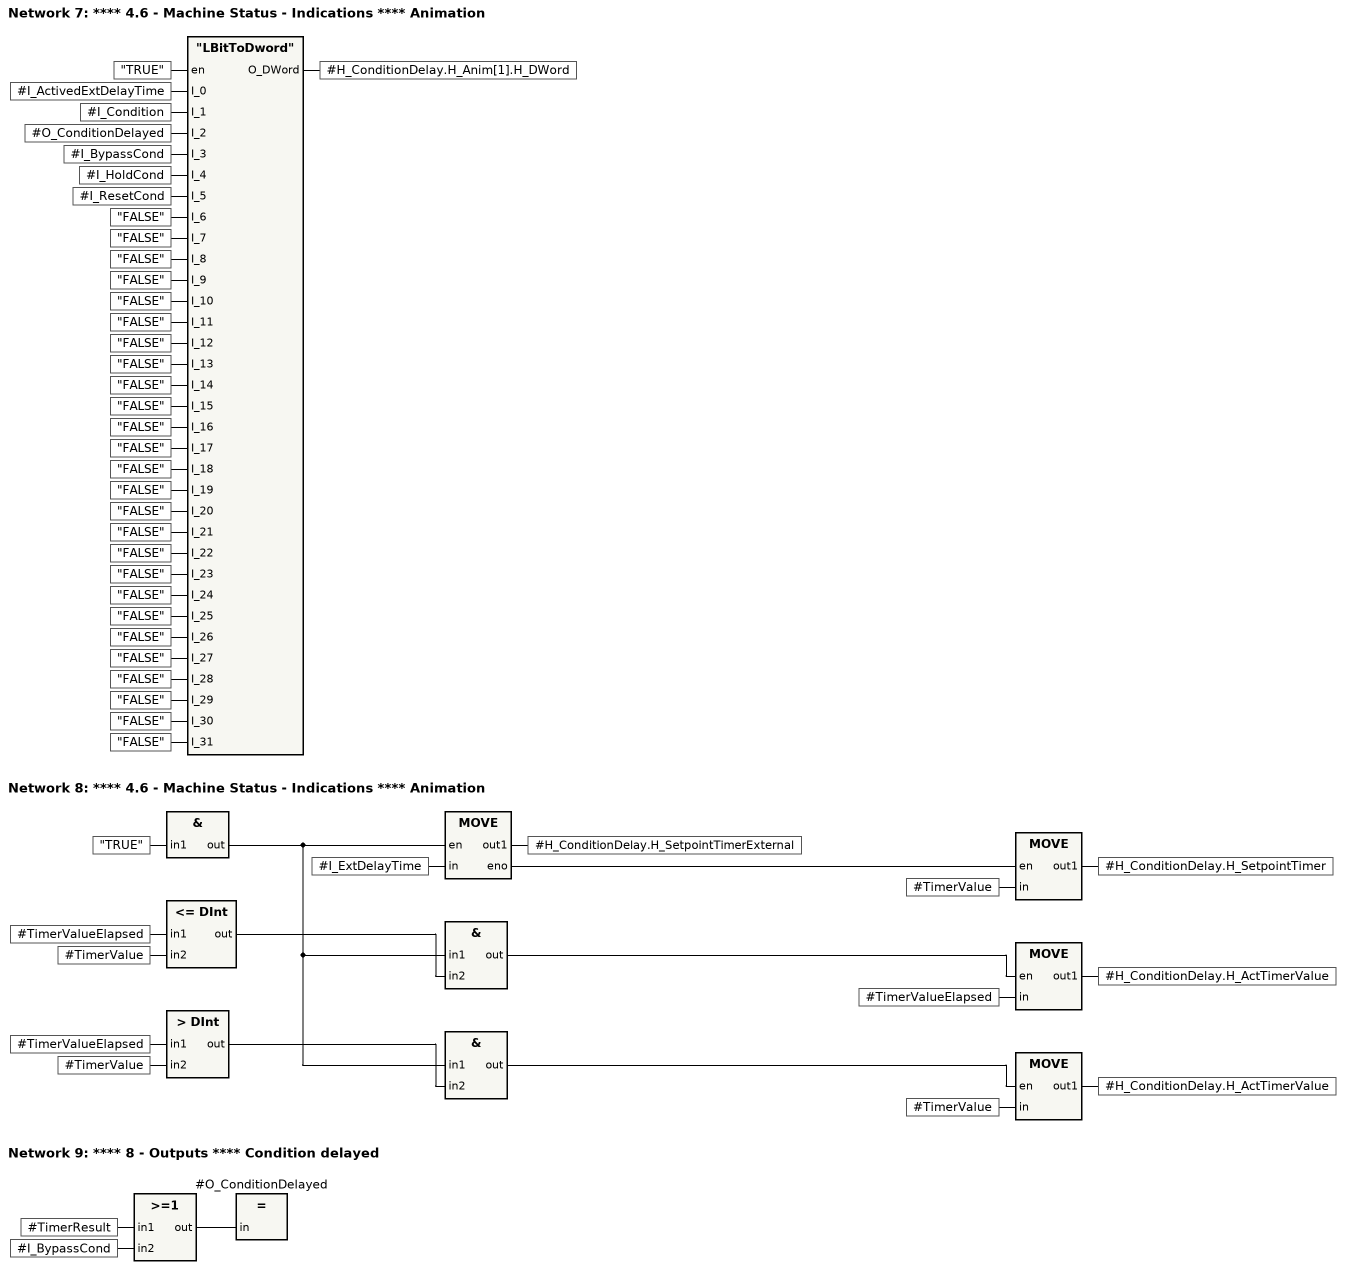
   IF "TRUE" THEN
       "LBitToDword"(I_0 := #I_ActivedExtDelayTime,
                     I_1 := #I_Condition,
                     I_2 := #O_ConditionDelayed,
                     I_3 := #I_BypassCond,
                     I_4 := #I_HoldCond,
                     I_5 := #I_ResetCond,
                     I_6 := "FALSE",
                     I_7 := "FALSE",
                     I_8 := "FALSE",
                     I_9 := "FALSE",
                     I_10 := "FALSE",
                     I_11 := "FALSE",
                     I_12 := "FALSE",
                     I_13 := "FALSE",
                     I_14 := "FALSE",
                     I_15 := "FALSE",
                     I_16 := "FALSE",
                     I_17 := "FALSE",
                     I_18 := "FALSE",
                     I_19 := "FALSE",
                     I_20 := "FALSE",
                     I_21 := "FALSE",
                     I_22 := "FALSE",
                     I_23 := "FALSE",
                     I_24 := "FALSE",
                     I_25 := "FALSE",
                     I_26 := "FALSE",
                     I_27 := "FALSE",
                     I_28 := "FALSE",
                     I_29 := "FALSE",
                     I_30 := "FALSE",
                     I_31 := "FALSE",
                     O_DWord => #H_ConditionDelay.H_Anim[1].H_DWord);
   END_IF;
END_REGION

REGION Network 8: **** 4.6 - Machine Status - Indications **** Animation
   IF "TRUE" THEN
       #H_ConditionDelay.H_SetpointTimerExternal := #I_ExtDelayTime;
       #H_ConditionDelay.H_SetpointTimer := #TimerValue;
   END_IF;
   IF "TRUE" AND (#TimerValueElapsed <= #TimerValue) THEN
       #H_ConditionDelay.H_ActTimerValue := #TimerValueElapsed;
   END_IF;
   IF "TRUE" AND (#TimerValueElapsed > #TimerValue) THEN
       #H_ConditionDelay.H_ActTimerValue := #TimerValue;
   END_IF;
END_REGION

REGION Network 9: **** 8 - Outputs **** Condition delayed
   #O_ConditionDelayed := #TimerResult OR #I_BypassCond;
END_REGION
END_FUNCTION_BLOCK

FUNCTION_BLOCK "LMovFnc2Pos"   // FB1102, FBD
TITLE = LMovFnc2Pos
{ S7_Optimized_Access := 'TRUE' }
AUTHOR : VCC
FAMILY : Tooling
VERSION : 0.1
// =============================================================================
// This module will be used for the steering of a two Position movement.
// It will get the commands from different Modes, evaluate the status of the 
// Interlock and give the command to the Actuator or direct to simple outputs.
// =============================================================================
// stored: AutoNumber false, IsIECCheckEnabled false, IsRetainMemResEnabled false, MemoryReserve 100, SetENOAutomatically False, UDAEnableTagReadback false
   VAR_INPUT
      I_PosSet { ExternalAccessible := 'False'; ExternalVisible := 'False'; ExternalWritable := 'False'} : Bool;   // Position Set detection or summary / Position Set Detection
      I_PosRes { ExternalAccessible := 'False'; ExternalVisible := 'False'; ExternalWritable := 'False'} : Bool;   // Position Reset detection or summary / Position Reset Detection
      I_PBSet { ExternalAccessible := 'False'; ExternalVisible := 'False'; ExternalWritable := 'False'} : Bool;   // Push button for Set direction (used in manual with button OP panels )
      I_PBReset { ExternalAccessible := 'False'; ExternalVisible := 'False'; ExternalWritable := 'False'} : Bool;   // Push button for reset direcion (used in manual with pushbutton OP panels) / Push button for Reset direction (used in manual with Pushbutton OP panels)
      I_SetBegin { ExternalAccessible := 'False'; ExternalVisible := 'False'; ExternalWritable := 'False'} : Bool;   // Function Set begin selection
      I_ResBegin { ExternalAccessible := 'False'; ExternalVisible := 'False'; ExternalWritable := 'False'} : Bool;   // Function Reset begin selection
      I_SetIntlkOK { ExternalAccessible := 'False'; ExternalVisible := 'False'; ExternalWritable := 'False'} : Bool;   // Set Interlock
      I_ResIntlkOK { ExternalAccessible := 'False'; ExternalVisible := 'False'; ExternalWritable := 'False'} : Bool;   // Reset Interlock
      I_SafetyOk { ExternalAccessible := 'False'; ExternalVisible := 'False'; ExternalWritable := 'False'} : Bool;   // Safety Ok
      I_HardwareOk { ExternalAccessible := 'False'; ExternalVisible := 'False'; ExternalWritable := 'False'} : Bool;   // Safety Ok / Hardware Ok
   END_VAR
   VAR_OUTPUT
      O_CmdSet { ExternalAccessible := 'False'; ExternalVisible := 'False'; ExternalWritable := 'False'} : Bool;   // Command to activate Set movement / Command to Activate Set movement
      O_CmdRes { ExternalAccessible := 'False'; ExternalVisible := 'False'; ExternalWritable := 'False'} : Bool;   // Command to activate Reset movement / Command to Activate Reset movement
      O_FuncRunning { ExternalAccessible := 'False'; ExternalVisible := 'False'; ExternalWritable := 'False'} : Bool;   // Signal that the function is running
      O_FuncBusyTM { ExternalAccessible := 'False'; ExternalVisible := 'False'; ExternalWritable := 'False'} : Bool;   // Memory Signal that the function is busy
      O_SetFinished { ExternalAccessible := 'False'; ExternalVisible := 'False'; ExternalWritable := 'False'} : Bool;   // Function Set finished to Master Sequencing
      O_ResFinished { ExternalAccessible := 'False'; ExternalVisible := 'False'; ExternalWritable := 'False'} : Bool;   // Function Reset finished to Master Sequencing
      O_IntlkSetAlm { ExternalAccessible := 'False'; ExternalVisible := 'False'; ExternalWritable := 'False'} : Bool;   // Alarm interlock Set / Alarm Interlock Set
      O_IntlkResAlm { ExternalAccessible := 'False'; ExternalVisible := 'False'; ExternalWritable := 'False'} : Bool;   // Alarm interlock Reset / Alarm Interlock Reset
      O_FuncIsSelInMan { ExternalAccessible := 'False'; ExternalVisible := 'False'; ExternalWritable := 'False'} : Bool;   // The function is selected in manual mode / The function is Selected in manual Mode
      O_LED { ExternalAccessible := 'False'; ExternalVisible := 'False'; ExternalWritable := 'False'} : Bool;   // LED-indication / LED - Indication
      O_AlarmABCondition { ExternalAccessible := 'False'; ExternalVisible := 'False'; ExternalWritable := 'False'} : Bool;   // Alarms AB condition / Alarm AB Condition
   END_VAR
   VAR_IN_OUT
      IO_Modes : "Modes";   // Modes
      H_HMI : "H_HMI";   // Animation
      H_MovFnc2Pos : "H_MovFnc2Pos";   // Animation
      H_FncSelInHMI { ExternalAccessible := 'False'; ExternalVisible := 'False'; ExternalWritable := 'False'} : Bool;   // This function is selected to run from HMI / This function is Selected to run from HMI
      C_AlarmResetUsed { ExternalAccessible := 'False'; ExternalVisible := 'False'; ExternalWritable := 'False'} : Bool;   // If true, the alrms will be stored untill reseted / If TRUE The Alarms will be stored untill Reseted
      C_EnableMemBegin { ExternalAccessible := 'False'; ExternalVisible := 'False'; ExternalWritable := 'False'} : Bool;   // Enable memory Begin (Command request is memorised until pos reached) / Enable memory Begin (Command Request is memorised until pos reached)
      C_EnIntlkAlm { ExternalAccessible := 'False'; ExternalVisible := 'False'; ExternalWritable := 'False'} : Bool := TRUE;   // Enable Interlock Alarm
      C_SetReset { ExternalAccessible := 'False'; ExternalVisible := 'False'; ExternalWritable := 'False'} : Bool;   // Enable Set Reset Functionality ( If enabled output is kept until the Cmd direction is changed )
      C_ManualClampCmdSet { ExternalAccessible := 'False'; ExternalVisible := 'False'; ExternalWritable := 'False'} : Bool;   // Manual Clamp Set
      C_ManualClampCmdRes { ExternalAccessible := 'False'; ExternalVisible := 'False'; ExternalWritable := 'False'} : Bool;   // Manual Clamp Reset
      C_ForceManual { ExternalAccessible := 'False'; ExternalVisible := 'False'; ExternalWritable := 'False'} : Bool := FALSE;   // Force Manual
   END_VAR
   VAR
      ResetAlarm { ExternalAccessible := 'False'; ExternalVisible := 'False'; ExternalWritable := 'False'} : Bool;   // Reset Alarm Memory
      CmdSetRequest { ExternalAccessible := 'False'; ExternalVisible := 'False'; ExternalWritable := 'False'} : Bool;   // Set Command request to activate the interlock / Set Command Request to Activate the Interlock
      CmdResRequest { ExternalAccessible := 'False'; ExternalVisible := 'False'; ExternalWritable := 'False'} : Bool;   // Reset Command request to activate the interlock / Reset Command Request to Activate the Interlock
      EdgeStopDetSet { ExternalAccessible := 'False'; ExternalVisible := 'False'; ExternalWritable := 'False'} : Bool;   // Edge on stop detection to be abble to go over it in force manual
      EdgeStopDetRes { ExternalAccessible := 'False'; ExternalVisible := 'False'; ExternalWritable := 'False'} : Bool;   // Edge on stop detection to be abble to go over it in force manual
      IntlkSetAlm { ExternalAccessible := 'False'; ExternalVisible := 'False'; ExternalWritable := 'False'} : Bool;   // Alarm interlock Set / Alarm Interlock Set
      IntlkResAlm { ExternalAccessible := 'False'; ExternalVisible := 'False'; ExternalWritable := 'False'} : Bool;   // Alarm interlock Reset / Alarm Interlock Reset
      CmdSet { ExternalAccessible := 'False'; ExternalVisible := 'False'; ExternalWritable := 'False'} : Bool;   // Command to activate Set movement / Command to Activate Set movement
      CmdRes { ExternalAccessible := 'False'; ExternalVisible := 'False'; ExternalWritable := 'False'} : Bool;   // Command to activate Reset movement / Command to Activate Reset movement
      IntlkSetAlmCond { ExternalAccessible := 'False'; ExternalVisible := 'False'; ExternalWritable := 'False'} : Bool;   // Alarm interlock Set condition / Alarm Interlock Set condition
      IntlkResAlmCond { ExternalAccessible := 'False'; ExternalVisible := 'False'; ExternalWritable := 'False'} : Bool;   // Alarm interlock Reset condition / Alarm Interlock Reset condition
      FuncRunning { ExternalAccessible := 'False'; ExternalVisible := 'False'; ExternalWritable := 'False'} : Bool;   // Function is running
      FuncBusyTM { ExternalAccessible := 'False'; ExternalVisible := 'False'; ExternalWritable := 'False'} : Bool;   // Memory Signal that the function is busy
      AlmFilterResult { ExternalAccessible := 'False'; ExternalVisible := 'False'; ExternalWritable := 'False'} : Bool;   // Alarm filter result
      _AlarmTimer { ExternalAccessible := 'False'; ExternalVisible := 'False'; ExternalWritable := 'False'} : "LTimer";
   END_VAR
   VAR_TEMP   // added for the SCL form of the ladder/FBD networks
      _w1 : Bool;
   END_VAR
BEGIN

REGION Network 1: **** 2.2 - Alarms - Alarm Generation **** Alarm Filter
   // Alarm Filter
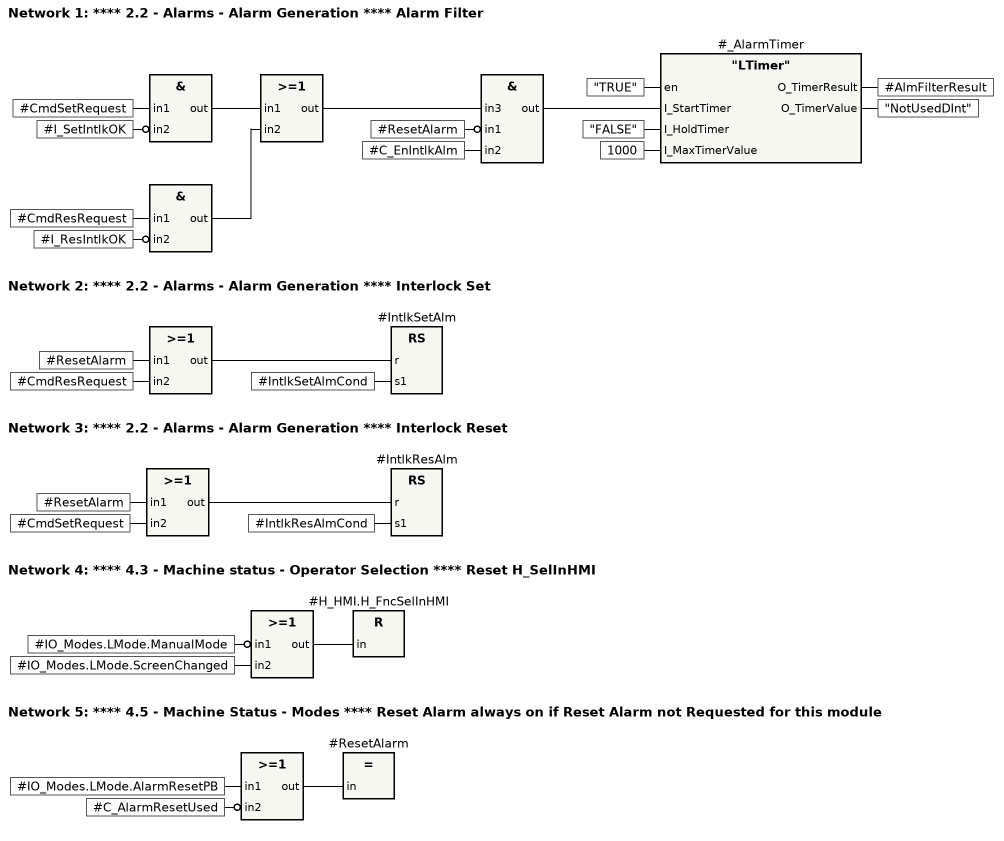
   IF "TRUE" THEN
       #_AlarmTimer(I_StartTimer := ((#CmdSetRequest AND NOT #I_SetIntlkOK) OR (#CmdResRequest AND NOT #I_ResIntlkOK)) AND NOT #ResetAlarm AND #C_EnIntlkAlm,   // "LTimer"
                    I_HoldTimer := "FALSE",
                    I_MaxTimerValue := 1000,
                    O_TimerResult => #AlmFilterResult,
                    O_TimerValue => "NotUsedDInt");
   END_IF;
END_REGION

REGION Network 2: **** 2.2 - Alarms - Alarm Generation **** Interlock Set
   // Interlock Set
   IF #ResetAlarm OR #CmdResRequest THEN
       #IntlkSetAlm := FALSE;   // RS flip-flop
   END_IF;
   IF #IntlkSetAlmCond THEN #IntlkSetAlm := TRUE; END_IF;
END_REGION

REGION Network 3: **** 2.2 - Alarms - Alarm Generation **** Interlock Reset
   // Interlock Reset
   IF #ResetAlarm OR #CmdSetRequest THEN
       #IntlkResAlm := FALSE;   // RS flip-flop
   END_IF;
   IF #IntlkResAlmCond THEN #IntlkResAlm := TRUE; END_IF;
END_REGION

REGION Network 4: **** 4.3 - Machine status - Operator Selection **** Reset H_SelInHMI
   // Reset H_SelInHMI
   IF NOT #IO_Modes.LMode.ManualMode OR #IO_Modes.LMode.ScreenChanged THEN
       #H_HMI.H_FncSelInHMI := FALSE;
   END_IF;
END_REGION

REGION Network 5: **** 4.5 - Machine Status - Modes **** Reset Alarm always on if Reset Alarm not Requested for this module
   // Reset Alarm always on if Reset Alarm not Requested for this module
   #ResetAlarm := #IO_Modes.LMode.AlarmResetPB OR NOT #C_AlarmResetUsed;
END_REGION

REGION Network 6: **** 4.6 - Machine Status - Indication **** Icon Animation
   // Icon Animation
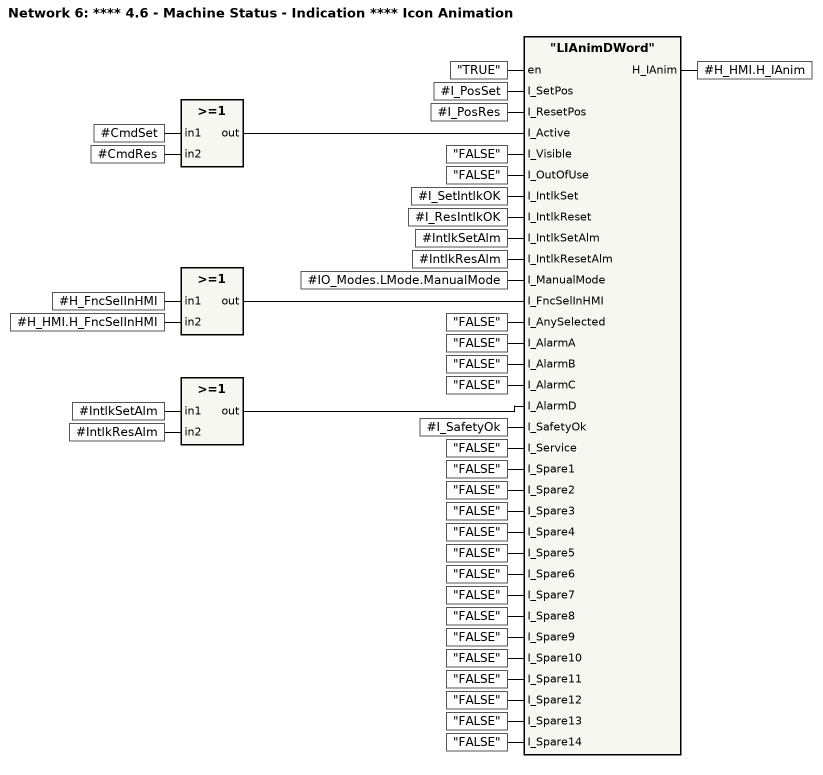
   IF "TRUE" THEN
       "LIAnimDWord"(I_SetPos := #I_PosSet,
                     I_ResetPos := #I_PosRes,
                     I_Active := #CmdSet OR #CmdRes,
                     I_Visible := "FALSE",
                     I_OutOfUse := "FALSE",
                     I_IntlkSet := #I_SetIntlkOK,
                     I_IntlkReset := #I_ResIntlkOK,
                     I_IntlkSetAlm := #IntlkSetAlm,
                     I_IntlkResetAlm := #IntlkResAlm,
                     I_ManualMode := #IO_Modes.LMode.ManualMode,
                     I_FncSelInHMI := #H_FncSelInHMI OR #H_HMI.H_FncSelInHMI,
                     I_AnySelected := "FALSE",
                     I_AlarmA := "FALSE",
                     I_AlarmB := "FALSE",
                     I_AlarmC := "FALSE",
                     I_AlarmD := #IntlkSetAlm OR #IntlkResAlm,
                     I_SafetyOk := #I_SafetyOk,
                     I_Service := "FALSE",
                     I_Spare1 := "FALSE",
                     I_Spare2 := "FALSE",
                     I_Spare3 := "FALSE",
                     I_Spare4 := "FALSE",
                     I_Spare5 := "FALSE",
                     I_Spare6 := "FALSE",
                     I_Spare7 := "FALSE",
                     I_Spare8 := "FALSE",
                     I_Spare9 := "FALSE",
                     I_Spare10 := "FALSE",
                     I_Spare11 := "FALSE",
                     I_Spare12 := "FALSE",
                     I_Spare13 := "FALSE",
                     I_Spare14 := "FALSE",
                     H_IAnim => #H_HMI.H_IAnim);
   END_IF;
END_REGION

REGION Network 7: **** 4.6 - Machine Status - Indication **** Animation
   // Animation
